# B&R Automation Studio project Agroittica (part 4)

```iecst
				intern.AsIOAccWriteValue := (51200/UINT_TO_REAL(intern.Parameters.Units_rev)) * (DINT_TO_REAL(IO_Cfg.MPGen.RefSpeed)/40.0);	(* Scale from units/s to uSteps/25ms. *)

				IF ((AsIOAccWrite_0.status = ERR_OK) AND ((intern.AsIOAccWriteValue > 65535.0) OR (intern.AsIOAccWriteValue < -65535.0) OR (* Overflow *)
	 					((IO_Cfg.MPGen.RefSpeed > 0) AND (intern.AsIOAccWriteValue < 0))) OR																					(* Positive overflow? *)
						((IO_Cfg.MPGen.RefSpeed < 0) AND (intern.AsIOAccWriteValue > 0))) THEN																				(* Negative overflow? *)

					IF ((intern.OverflowWarning > 1_00_00_00) OR (intern.OverflowWarning < 0)) THEN																	(* Already recorded 4 overflow states? *)
						intern.OverflowWarning := ((ABS(intern.OverflowWarning) + 1_00_00_00_00) * -1);																(* Make number negative and show number of overflow's occured + 4 recorded. *)
					ELSE
						intern.OverflowWarning := (intern.OverflowWarning * 100) + intern.StateMan;																		(* Recorded which step where overflow occured. *)
					END_IF

					IF (IO_Cfg.MPGen.RefSpeed > 0) THEN																																							(* Positive overflow? *)
						AsIOAccWrite_0.value := 65535;																																								(* Set to maximum. (16#FFFF = 65535) *)
					ELSIF (IO_Cfg.MPGen.RefSpeed < 0) THEN																																					(* Negitive overflow? *)
						AsIOAccWrite_0.value := -65535;																																								(* Set to maximum. (16# = -65535) *)
					END_IF

				ELSE																																																							(* Write value not overflowed. *)
					AsIOAccWrite_0.value := REAL_TO_UDINT(intern.AsIOAccWriteValue);																								(* Copy required write value. *)
				END_IF

				AsIOAccWrite_0(enable:=1, pDeviceName:=ADR(intern.IO_Mapping.DeviceName), pChannelName:=ADR(intern.ChannelName));	(* Write to register. *)

				IF (AsIOAccWrite_0.status <> ERR_FUB_BUSY) THEN																																		(* Function done? *)
					IF (AsIOAccWrite_0.status = ERR_OK) THEN																																				(* No error? *)

						IF ((Mode = 0) OR (Mode = 60) OR (intern.Cfg_State = 255)) THEN																								(* Write all configuration values to XMS module? *)
							intern.StateMan := intern.StateMan + 1;																																			(* Next XSM step. *)
						ELSE
							Done						:= 1;																																												(* Set Done flag. *)
							intern.StateMan := 0;																																												(* Wait for new command. *)
						END_IF

					ELSE																																																						(* AsIOAccRead Error? *)
						Status					:= AsIOAccWrite_0.status;																																			(* Copy AsIOAccWrite status. *)
					END_IF
				END_IF
			#endif
			#ifdef _SGC
				CASE (intern.IO_Mapping.Channel) OF
					0..1:		AsIOAccWriteReg_0.registerNr:= 68;																																			(* 1st motor channel selected. (Reg 68) *)
					2:			AsIOAccWriteReg_0.registerNr:= 132;																																			(* 2nd motor channel selected. (Reg 132) *)
					3:			AsIOAccWriteReg_0.registerNr:= 196;																																			(* 3rd motor channel selected. (Reg 196) *)
					4:			AsIOAccWriteReg_0.registerNr:= 260;																																			(* 4th motor channel selected. (Reg 260) *)
				END_CASE

				intern.AsIOAccWriteValue := (51200/UINT_TO_REAL(intern.Parameters.Units_rev)) * (DINT_TO_REAL(IO_Cfg.MPGen.RefSpeed)/40.0);	(* Scale from units/s to uSteps/25ms. *)

				IF ((AsIOAccWrite_0.status = ERR_OK) AND ((intern.AsIOAccWriteValue > 65535.0) OR (intern.AsIOAccWriteValue < -65535.0) OR (* Overflow *)
	 					((IO_Cfg.MPGen.RefSpeed > 0) AND (intern.AsIOAccWriteValue < 0))) OR																					(* Positive overflow? *)
						((IO_Cfg.MPGen.RefSpeed < 0) AND (intern.AsIOAccWriteValue > 0))) THEN																				(* Negative overflow? *)

					IF ((intern.OverflowWarning > 1_00_00_00) OR (intern.OverflowWarning < 0)) THEN																	(* Already recorded 4 overflow states? *)
						intern.OverflowWarning := ((ABS(intern.OverflowWarning) + 1_00_00_00_00) * -1);																(* Make number negative and show number of overflow's occured + 4 recorded. *)
					ELSE
						intern.OverflowWarning := (intern.OverflowWarning * 100) + intern.StateMan;																		(* Recorded which step where overflow occured. *)
					END_IF

					IF (IO_Cfg.MPGen.RefSpeed > 0) THEN																																							(* Positive overflow? *)
						AsIOAccWriteReg_0.value := 65535;																																							(* Set to maximum. (16#FFFF = 65535) *)
					ELSIF (IO_Cfg.MPGen.RefSpeed < 0) THEN																																					(* Negitive overflow? *)
						AsIOAccWriteReg_0.value := -65535;																																						(* Set to maximum. (16# = -65535) *)
					END_IF

				ELSE																																																							(* Write value not overflowed. *)
					AsIOAccWriteReg_0.value := REAL_TO_UDINT(intern.AsIOAccWriteValue);																							(* Copy required write value. *)
				END_IF

				AsIOAccWriteReg_0(enable:=1, size:=2);																																						(* Write to register. *)

				IF (AsIOAccWriteReg_0.status <> ERR_FUB_BUSY) THEN																																(* Function done? *)
					IF (AsIOAccWriteReg_0.status = ERR_OK) THEN																																			(* No error? *)

						IF ((Mode = 0) OR (Mode = 60) OR (intern.Cfg_State = 255)) THEN																								(* Write all configuration values to XMS module? *)
							intern.StateMan := intern.StateMan + 1;																																			(* Next XSM step. *)
						ELSE
							Done						:= 1;																																												(* Set Done flag. *)
							intern.StateMan := 0;																																												(* Wait for new command. *)
						END_IF

					ELSIF ((AsIOAccWriteReg_0.status = ioacERR_ACCESS) AND (intern.Retries < 2)) THEN																(* Access error? try again upto 2 times. *)
						intern.Retries:= intern.Retries + 1;																																					(* Increament retries counter. *)
					ELSE																																																						(* AsIOAccRead Error? *)
						Status					:= AsIOAccWriteReg_0.status;																																	(* Copy AsIOAccWrite status. *)
					END_IF
				END_IF
			#endif

			(* IO Configuration - Jolt time limitation. *)
			67:
				IF (IO_Cfg.MPGen.JoltTimeLimitation > 16) THEN																																		(* Jolt Time Limitation invalid? *)

					Status := 50267;																																																(* JoltTimeLimitation_Invalid *)

				ELSE

				#ifdef _SG4
					CASE (intern.IO_Mapping.Channel) OF
						0..1:		intern.ChannelName := 'JoltTime01';																																		(* 1st motor channel selected. (Reg 75) *)
						2:			intern.ChannelName := 'JoltTime02';																																		(* 2nd motor channel selected. (Reg 139) *)
						3:			intern.ChannelName := 'JoltTime03';																																		(* 3rd motor channel selected. (Reg 203) *)
						4:			intern.ChannelName := 'JoltTime04';																																		(* 4th motor channel selected. (Reg 267) *)
					END_CASE

					AsIOAccWrite_0.value := SINT_TO_UDINT(IO_Cfg.MPGen.JoltTimeLimitation);																					(* Required value. *)
					AsIOAccWrite_0(enable:=1, pDeviceName:=ADR(intern.IO_Mapping.DeviceName), pChannelName:=ADR(intern.ChannelName));	(* Write to register. *)

					IF (AsIOAccWrite_0.status <> ERR_FUB_BUSY) THEN																																	(* Function done? *)
						IF (AsIOAccWrite_0.status = ERR_OK) THEN																																			(* No error? *)
							IF ((Mode = 0) OR (Mode = 60) OR (intern.Cfg_State = 255)) THEN																							(* Module power back on? *)
								intern.Cfg_State := 1;																																										(* Reset IO Cfg Done flag. *)
							END_IF
							Done						:= 1;																																												(* Set Done flag. *)
							intern.StateMan := 0;																																												(* Wait for new command. *)
						ELSE																																																					(* AsIOAccRead Error? *)
							Status					:= AsIOAccWrite_0.status;																																		(* Copy AsIOAccWrite status. *)
						END_IF
					END_IF
				#endif
				#ifdef _SGC
					CASE (intern.IO_Mapping.Channel) OF
						0..1:		AsIOAccWriteReg_0.registerNr:= 75;																																		(* 1st motor channel selected. (Reg 75) *)
						2:			AsIOAccWriteReg_0.registerNr:= 139;																																		(* 2nd motor channel selected. (Reg 139) *)
						3:			AsIOAccWriteReg_0.registerNr:= 203;																																		(* 3rd motor channel selected. (Reg 203) *)
						4:			AsIOAccWriteReg_0.registerNr:= 267;																																		(* 4th motor channel selected. (Reg 267) *)
					END_CASE

					AsIOAccWriteReg_0.value := SINT_TO_UDINT(IO_Cfg.MPGen.JoltTimeLimitation);																			(* Required value. *)
					AsIOAccWriteReg_0(enable:=1, size:=1);																																					(* Write to register. *)

					IF (AsIOAccWriteReg_0.status <> ERR_FUB_BUSY) THEN																															(* Function done? *)
						IF (AsIOAccWriteReg_0.status = ERR_OK) THEN																																		(* No error? *)
							IF ((Mode = 0) OR (Mode = 60) OR (intern.Cfg_State = 255)) THEN																							(* Module power back on? *)
								intern.Cfg_State := 1;																																										(* Reset IO Cfg Done flag. *)
							END_IF
							Done						:= 1;																																												(* Set Done flag. *)
							intern.StateMan := 0;																																												(* Wait for new command. *)
						ELSIF ((AsIOAccWriteReg_0.status = ioacERR_ACCESS) AND (intern.Retries < 2)) THEN															(* Access error? try again upto 2 times. *)
							intern.Retries:= intern.Retries + 1;																																				(* Increament retries counter. *)
						ELSE																																																					(* AsIOAccRead Error? *)
							Status					:= AsIOAccWrite_0.status;																																		(* Copy AsIOAccWrite status. *)
						END_IF
					END_IF
				#endif

				END_IF

			(* Error handling - Check reset flag is OFF. *)
			1000:

				IF (pIO_Mapping <> 0) THEN																																												(* Address non-Zero? *)
					memcpy(ADR(intern.IO_Mapping), pIO_Mapping, SIZEOF(intern.IO_Mapping));																					(* Get update intern.IO_Mapping data. *)
				ELSE																																																							(* Error? *)
					Status := 50202;																																																(* pintern.IO_Mapping_Invalid. *)
				END_IF

				IF ((intern.Cfg_State = 255) AND (intern.IO_Mapping.ModuleOK)) THEN																								(* Module power back on? *)
					Status						:= 0;																																													(* Reset status. *)
					intern.StateMan 	:= 0;																																													(* Wait for new command. *)
				ELSIF (NOT(Reset) AND (intern.Cfg_State <> 255))THEN																															(* Reset OFF? *)
					intern.StateMan := intern.StateMan + 1;																																					(* Next XSM step. *)
				END_IF

			(* Error handling - Reset error on positve edge. *)
			1001:

				IF (Reset) THEN																																																		(* Reset / Error acknownledge? *)
					Reset							:= 0;																																													(* Reset reset. *)
					Status						:= 0;																																													(* Reset status. *)
				END_IF

				IF (NOT(Config) AND (Status = 0)) THEN																																						(* Start new configuration reset? *)
					intern.StateMan 	:= 0;																																													(* Wait for new command. *)
				END_IF

			(* Should not get here, invalid state. *)
			ELSE
				intern.StateMan := 1000;

		END_CASE

	ELSE
		intern.StateMan 	:= 0;																																																(* Wait for new command. *)
		Status := ERR_FUB_ENABLE_FALSE;																																												(* Function not enabled status. *)
	END_IF

	(********************************************************************************************************************
		!!!!!!!!!!!!!!!!!!!!!!!!!!!!!!!!!!!!!!!!! NO MORE CODE BEYOND THIS POINT !!!!!!!!!!!!!!!!!!!!!!!!!!!!!!!!!!!!!!!!!
	*********************************************************************************************************************)
END_FUNCTION_BLOCK
```

#### XSM_AcyclicRead.st - Provide alarm detail in form of BOOLEAN array for VC & User.
```iecst
FUNCTION_BLOCK XSM_AcyclicRead
	(* Implementation of XSM_AcyclicRead *)
	(********************************************************************************************************************
		Filename		: XSM_AcyclicRead.scr
		Version			: 00.01
		Date				: 14th July 2009
		Written by	: Andy Lees at B&R Industrial Automation Ltd. (UK)
		Customer		: Sheepy.
		Application : .
		Description	:	Provide alarm detail in form of BOOLEAN array for VC & User.

									Status:-

										0				ERR_OK

										50100		XSM_ModuleNotOK
										50101		XSM_ModuleID_Invalid -	X20 ->	X20SM1426 = 9857,						1x Stepper motor module 1A, 4 DI
																														X20SM1436 = 9858,						1x Stepper motor module 3A, 4 DI

																										X67 ->	X67SM2436 = 7627,						2x Stepper motor module 3A, 2x3 DI
																														X67SM4320 = 7628,						4x Stepper motor module 1A

																						ACOPOSmicro ->	80SD100XD.C0XX-01 = 42148,	2x Stepper motor 10 A, X2X, 2 Trigger Inputs.
																														80SD100XS.C0XX-01 = 42414,	1x Stepper motor 10 A, X2X, 2 DI (1 Trigger Input).
 																														80SD100XS.C04X-01 = 42880,	1x Stepper motor 10 A, X2X, 2 DI (1 Trigger Input), 1x ABR.
																														80SD100XD.C044-01 = 42881,	2x Stepper motor 10 A, X2X, 2x ABR, 2 Trigger Inputs.
																														80SD100XS.C04X-13 = 42882,	1x Stepper motor 10 A, X2X, 1x ABR, 4 DI/2 DO
																														80SD100XD.C04X-13 = 42893,	2x Stepper motor 10 A, X2X, 1x ABR, 4 DI/2 DO.
																														80SD100XD.C0XX-21 = 42894,	2x Stepper motor 10 A, X2X, 2 Inputs ±10 V.
										50109		XSM_Motor_Invalid.

										50202		pIO_Mapping_Invalid.

										50200		Read acyclic mode invalid.

										30190 - 30199 AsIOAcc

										65534		ERR_FUB_ENABLE_FALSE

									Mode:-

										1				Read DC bus voltage in V.
										2				Read Module temperature of the power output stage in °C.
										3				Read Module temperature in °C.

										4				Read Referenced zero position of the cyclic counter.
										5				Read Current position acyclic.
										6				Read Referenced zero position of the acyclic counter.

		History			: 14th July 2009		v00.01
									First release - Tested on X20CP1486 N2.95 with X20SM1426 on X2X & Ethernet Power Link.

	*********************************************************************************************************************)
	IF (Enable) THEN																																																			(* Function block enabled? *)

		(******************************************************************************************************************
			Errors force to handle errors?
		*******************************************************************************************************************)
		IF ((Status <> ERR_OK) AND (Status <> ERR_FUB_ENABLE_FALSE) AND (Status <> ERR_FUB_BUSY) AND (intern.StateMan < 1000)) THEN	(* Error and not error handling state's? *)
			intern.StateMan := 1000;																																														(* Handle errors. *)
		END_IF

		(******************************************************************************************************************
			SXM IO Configuratin state machine.
		*******************************************************************************************************************)
		CASE (intern.StateMan) OF																																															(* State machine. *)

			(* Init - Wait for command. *)
			0:
				IF ((Status = ERR_FUB_ENABLE_FALSE) OR (Status = ERR_FUB_BUSY)) THEN																							(* Clear function not enable or busy status? *)
					Status := ERR_OK;																																																(* Function OK. *)
				END_IF

				IF (pIO_Mapping <> 0) THEN																																												(* Address non-Zero? *)
					memcpy(ADR(intern.IO_Mapping), pIO_Mapping, SIZEOF(intern.IO_Mapping));																					(* Get update intern.IO_Mapping data. *)
				ELSE																																																							(* Error? *)
					Status := 50202;																																																(* pIO_Mapping_Invalid. *)
				END_IF

				IF ((intern.IO_Mapping.ModuleID <> 9857) AND (intern.IO_Mapping.ModuleID <> 9858) AND															(* Not X20SM1426, X20SM1436? *)
						(intern.IO_Mapping.ModuleID <> 7627) AND (intern.IO_Mapping.ModuleID <> 7628) AND															(* Not X67SM2436, X67SM4320? *)
						(intern.IO_Mapping.ModuleID <> 42148) AND (intern.IO_Mapping.ModuleID <> 42414) AND														(* Not 80SD100XD.C0XX-01, 80SD100XS.C0XX-01? *)
						(intern.IO_Mapping.ModuleID <> 42880) AND (intern.IO_Mapping.ModuleID <> 42881) AND														(* Not 80SD100XS.C04X-01, 80SD100XD.C044-01? *)
						(intern.IO_Mapping.ModuleID <> 42882) AND (intern.IO_Mapping.ModuleID <> 42893) AND														(* Not 80SD100XS.C04X-13, 80SD100XD.C04X-13? *)
						(intern.IO_Mapping.ModuleID <> 42894)) THEN																																		(* Not 80SD100XD.C0XX-21? *)
					Status := 50101;																																																(* Error - XSM_ModuleID_Invalid *)
				ELSIF (((intern.IO_Mapping.ModuleID = 9857) AND ((intern.IO_Mapping.Channel < 0) OR (intern.IO_Mapping.Channel > 1))) OR	(* X20SM1426 - Only 1 motor possible. *)
							 ((intern.IO_Mapping.ModuleID = 9858) AND ((intern.IO_Mapping.Channel < 0) OR (intern.IO_Mapping.Channel > 1))) OR	(* X20SM1436 - Only 1 motor possible. *)
							 ((intern.IO_Mapping.ModuleID = 7627) AND ((intern.IO_Mapping.Channel < 0) OR (intern.IO_Mapping.Channel > 2))) OR	(* X67SM2436 - Only 2 motor possible. *)
							 ((intern.IO_Mapping.ModuleID = 7628) AND ((intern.IO_Mapping.Channel < 0) OR (intern.IO_Mapping.Channel > 4)))	OR	(* X67SM4320 - Only 4 motor possible. *)
							 ((intern.IO_Mapping.ModuleID = 42148) AND ((intern.IO_Mapping.Channel < 0) OR (intern.IO_Mapping.Channel > 2))) OR	(* 80SD100XD.C0XX-01 - Only 2 motor possible. *)
							 ((intern.IO_Mapping.ModuleID = 42414) AND ((intern.IO_Mapping.Channel < 0) OR (intern.IO_Mapping.Channel > 1))) OR	(* 80SD100XS.C0XX-01 - Only 1 motor possible. *)
							 ((intern.IO_Mapping.ModuleID = 42880) AND ((intern.IO_Mapping.Channel < 0) OR (intern.IO_Mapping.Channel > 1))) OR	(* 80SD100XS.C04X-01 - Only 1 motor possible. *)
							 ((intern.IO_Mapping.ModuleID = 42881) AND ((intern.IO_Mapping.Channel < 0) OR (intern.IO_Mapping.Channel > 2))) OR	(* 80SD100XD.C044-01 - Only 2 motor possible. *)
							 ((intern.IO_Mapping.ModuleID = 42882) AND ((intern.IO_Mapping.Channel < 0) OR (intern.IO_Mapping.Channel > 1))) OR	(* 80SD100XS.C04X-13 - Only 1 motor possible. *)
							 ((intern.IO_Mapping.ModuleID = 42893) AND ((intern.IO_Mapping.Channel < 0) OR (intern.IO_Mapping.Channel > 2))) OR	(* 80SD100XD.C04X-13 - Only 2 motor possible. *)
							 ((intern.IO_Mapping.ModuleID = 42894) AND ((intern.IO_Mapping.Channel < 0) OR (intern.IO_Mapping.Channel > 2)))		(* 80SD100XD.C0XX-21 - Only 2 motor possible. *)
							) THEN																																																				(* Selected motor invalid? *)
					Status := 50109;																																																	(* XSM_Motor_Invalid? *)
				END_IF

			#ifdef _SGC
				AsIOAccReadReg_0.nodeNr:= DINT_TO_USINT(atoi(ADR(intern.IO_Mapping.DeviceName) + FIND(intern.IO_Mapping.DeviceName, 'ST') + 1));	(* Get node number on X2X. *)
			#endif

				intern.ReadOK:= (intern.ReadOK AND Read);																																				(* Detect +edge of Read. *)

				IF ((Status = ERR_OK) AND NOT(intern.ReadOK) AND (Read)) THEN																										(* Read acyclic data? *)
					intern.Retries:= 0;																																														(* Reset retries. *)
					Status := ERR_FUB_BUSY;																																												(* Function busy status. *)
					CASE (Mode) OF
						1:			intern.StateMan		:= 10;																																						(* Read DC bus voltage in V. *)
						2:			intern.StateMan 	:= 20;																																						(* Read Module temperature of the power output stage in °C. *)
						3:			intern.StateMan 	:= 30;																																						(* Read Module temperature in °C. *)
						4:			intern.StateMan 	:= 40;																																						(* Read Referenced zero position of the cyclic counter. *)
						5:			intern.StateMan 	:= 50;																																						(* Read Current position acyclic. *)
						6:			intern.StateMan 	:= 60;																																						(* Read Referenced zero position of the acyclic counter. *)
						ELSE	Status := 50400;																																											(* Read acyclic mode invalid. *)
					END_CASE
				END_IF

			(* Read DC bus voltage in V. *)
			10:
			#ifdef _SG4
				intern.ChannelName := 'UZKVoltage';																																							(* Read DC bus voltage in V. (Reg 42) *)

				AsIOAccRead_0(enable:=1, pDeviceName:=ADR(intern.IO_Mapping.DeviceName), pChannelName:=ADR(intern.ChannelName));	(* Read acyclic data. *)

				IF (AsIOAccRead_0.status <> ERR_FUB_BUSY) THEN																																	(* Function done? *)
					IF (AsIOAccRead_0.status = ERR_OK) THEN																																				(* No error? *)
						ReadData.DC_BusVoltage:= UDINT_TO_UINT(AsIOAccRead_0.value);																								(* Copy data. *)
						intern.ReadOK:= 	TRUE;																																											(* Read OK. *)
						intern.StateMan:= 0;
					ELSE																																																					(* AsIOAccRead Error? *)
						Status:= AsIOAccRead_0.status;
					END_IF
				END_IF
			#endif
			#ifdef _SGC
				AsIOAccReadReg_0.registerNr:= 42;																																								(* Read DC bus voltage in V. (Reg 42) *)

				AsIOAccReadReg_0(enable:= 1, size:= 2);																																					(* Read acyclic data. *)

				IF (AsIOAccReadReg_0.status <> ERR_FUB_BUSY) THEN																																(* Function done? *)
					IF (AsIOAccReadReg_0.status = ERR_OK) THEN																																		(* No error? *)
						ReadData.DC_BusVoltage:= UDINT_TO_UINT(AsIOAccReadReg_0.value);																							(* Update error code. *)
						intern.ReadOK:= 	TRUE;																																											(* Read OK. *)
						intern.StateMan:= 0;
					ELSIF ((AsIOAccReadReg_0.status = ioacERR_ACCESS) AND (intern.Retries < 2)) THEN															(* Access error? try again upto 2 times. *)
						intern.Retries:= intern.Retries + 1;																																				(* Increament retries counter. *)
					ELSE																																																					(* AsIOAccReadReg Error? *)
						Status:= AsIOAccReadReg_0.status;																																						(* Copy AsIOAccReadReg status. *)
					END_IF
				END_IF
			#endif

			(* Read Module temperature of the power output stage in °C. *)
			20:
			#ifdef _SG4
				intern.ChannelName := 'CoolerTemperature';																																			(* Read Module temperature of the power output stage in °C. (Reg 44) *)

				AsIOAccRead_0(enable:=1, pDeviceName:=ADR(intern.IO_Mapping.DeviceName), pChannelName:=ADR(intern.ChannelName));	(* Read acyclic data. *)

				IF (AsIOAccRead_0.status <> ERR_FUB_BUSY) THEN																																	(* Function done? *)
					IF (AsIOAccRead_0.status = ERR_OK) THEN																																				(* No error? *)
						ReadData.PowerStage_Temperature:= UDINT_TO_SINT(AsIOAccRead_0.value);																				(* Copy data. *)
						intern.ReadOK:= 	TRUE;																																											(* Read OK. *)
						intern.StateMan:= 0;
					ELSE																																																					(* AsIOAccRead Error? *)
						Status:= AsIOAccRead_0.status;
					END_IF
				END_IF
			#endif
			#ifdef _SGC
				AsIOAccReadReg_0.registerNr:= 44;																																								(* Read Module temperature of the power output stage in °C. (Reg 44). *)

				AsIOAccReadReg_0(enable:= 1, size:= 1);																																					(* Read acyclic data. *)

				IF (AsIOAccReadReg_0.status <> ERR_FUB_BUSY) THEN																																(* Function done? *)
					IF (AsIOAccReadReg_0.status = ERR_OK) THEN																																		(* No error? *)
						ReadData.PowerStage_Temperature:= UDINT_TO_SINT(AsIOAccReadReg_0.value);																		(* Update error code. *)
						intern.ReadOK:= 	TRUE;																																											(* Read OK. *)
						intern.StateMan:= 0;
					ELSIF ((AsIOAccReadReg_0.status = ioacERR_ACCESS) AND (intern.Retries < 2)) THEN															(* Access error? try again upto 2 times. *)
						intern.Retries:= intern.Retries + 1;																																				(* Increament retries counter. *)
					ELSE																																																					(* AsIOAccReadReg Error? *)
						Status:= AsIOAccReadReg_0.status;																																						(* Copy AsIOAccReadReg status. *)
					END_IF
				END_IF
			#endif

			(* Read Module temperature in °C. *)
			30:
			#ifdef _SG4
				intern.ChannelName := 'Temperature';																																						(* Read Module temperature in °C. (Reg 46) *)

				AsIOAccRead_0(enable:=1, pDeviceName:=ADR(intern.IO_Mapping.DeviceName), pChannelName:=ADR(intern.ChannelName));	(* Read acyclic data. *)

				IF (AsIOAccRead_0.status <> ERR_FUB_BUSY) THEN																																	(* Function done? *)
					IF (AsIOAccRead_0.status = ERR_OK) THEN																																				(* No error? *)
						ReadData.Module_Temperature:= UDINT_TO_SINT(AsIOAccRead_0.value);																						(* Copy data. *)
						intern.ReadOK:= 	TRUE;																																											(* Read OK. *)
						intern.StateMan:= 0;
					ELSE																																																					(* AsIOAccRead Error? *)
						Status:= AsIOAccRead_0.status;
					END_IF
				END_IF
			#endif
			#ifdef _SGC
				AsIOAccReadReg_0.registerNr:= 46;																																								(* Read Module temperature in °C. (Reg 46). *)

				AsIOAccReadReg_0(enable:= 1, size:= 1);																																					(* Read acyclic data. *)

				IF (AsIOAccReadReg_0.status <> ERR_FUB_BUSY) THEN																																(* Function done? *)
					IF (AsIOAccReadReg_0.status = ERR_OK) THEN																																		(* No error? *)
						ReadData.Module_Temperature:= UDINT_TO_SINT(AsIOAccReadReg_0.value);																				(* Update error code. *)
						intern.ReadOK:= 	TRUE;																																											(* Read OK. *)
						intern.StateMan:= 0;
					ELSIF ((AsIOAccReadReg_0.status = ioacERR_ACCESS) AND (intern.Retries < 2)) THEN															(* Access error? try again upto 2 times. *)
						intern.Retries:= intern.Retries + 1;																																				(* Increament retries counter. *)
					ELSE																																																					(* AsIOAccReadReg Error? *)
						Status:= AsIOAccReadReg_0.status;																																						(* Copy AsIOAccReadReg status. *)
					END_IF
				END_IF
			#endif

			(* Read Referenced zero position of the cyclic counter. *)
			40:
			#ifdef _SG4
				CASE (intern.IO_Mapping.Channel) OF
					0..1:		intern.ChannelName := 'RefPos01CyclicCounter';																												(* X20SM/X67SM/ACOPOSmicro 1st motor selected.(Reg 86)*)
					2:			intern.ChannelName := 'RefPos02CyclicCounter';																												(* X67SM/ACOPOSmicro 2nd motor selected. (Reg 150)*)
					3:			intern.ChannelName := 'RefPos03CyclicCounter';																												(* 3rd motor channel selected. (Reg 214) *)
					4:			intern.ChannelName := 'RefPos04CyclicCounter';																												(* 4th motor channel selected. (Reg 278) *)
				END_CASE

				AsIOAccRead_0(enable:=1, pDeviceName:=ADR(intern.IO_Mapping.DeviceName), pChannelName:=ADR(intern.ChannelName));	(* Read acyclic data. *)

				IF (AsIOAccRead_0.status <> ERR_FUB_BUSY) THEN																																	(* Function done? *)
					IF (AsIOAccRead_0.status = ERR_OK) THEN																																				(* No error? *)
						ReadData.Encoder_RefPosCyclicCounter:= UDINT_TO_DINT(AsIOAccRead_0.value);																	(* Copy data. *)
						intern.ReadOK:= 	TRUE;																																											(* Read OK. *)
						intern.StateMan:= 0;
					ELSE																																																					(* AsIOAccRead Error? *)
						Status:= AsIOAccRead_0.status;
					END_IF
				END_IF
			#endif
			#ifdef _SGC
				CASE (intern.IO_Mapping.Channel) OF
					0..1:		AsIOAccReadReg_0.registerNr:= 86;																																			(* X20SM/X67SM/ACOPOSmicro 1st motor selected.(Reg 86)*)
					2:			AsIOAccReadReg_0.registerNr:= 150;																																		(* X67SM/ACOPOSmicro 2nd motor selected. (Reg 150)*)
					3:			AsIOAccReadReg_0.registerNr:= 214;																																		(* 3rd motor channel selected. (Reg 214) *)
					4:			AsIOAccReadReg_0.registerNr:= 278;																																		(* 4th motor channel selected. (Reg 278) *)
				END_CASE

				AsIOAccReadReg_0(enable:= 1, size:= 4);																																					(* Read acyclic data. *)

				IF (AsIOAccReadReg_0.status <> ERR_FUB_BUSY) THEN																																(* Function done? *)
					IF (AsIOAccReadReg_0.status = ERR_OK) THEN																																		(* No error? *)
						ReadData.Encoder_RefPosCyclicCounter:= UDINT_TO_DINT(AsIOAccReadReg_0.value);																(* Update error code. *)
						intern.ReadOK:= 	TRUE;																																											(* Read OK. *)
						intern.StateMan:= 0;
					ELSIF ((AsIOAccReadReg_0.status = ioacERR_ACCESS) AND (intern.Retries < 2)) THEN															(* Access error? try again upto 2 times. *)
						intern.Retries:= intern.Retries + 1;																																				(* Increament retries counter. *)
					ELSE																																																					(* AsIOAccReadReg Error? *)
						Status:= AsIOAccReadReg_0.status;																																						(* Copy AsIOAccReadReg status. *)
					END_IF
				END_IF
			#endif

			(* Read Current position acyclic. *)
			50:
			#ifdef _SG4
				CASE (intern.IO_Mapping.Channel) OF
					0..1:		intern.ChannelName := 'AbsPos1ActValAcyclic';																												(* X20SM/X67SM/ACOPOSmicro 1st motor selected.(Reg 90)*)
					2:			intern.ChannelName := 'AbsPos2ActValAcyclic';																												(* X67SM/ACOPOSmicro 2nd motor selected. (Reg 154)*)
(*					3:			intern.ChannelName := 'AbsPos3ActValAcyclic';	- Not used yet *)																											(* 3rd motor channel selected. (Reg ???) *)
(*					4:			intern.ChannelName := 'AbsPos4ActValAcyclic';	- Not used yet *)																												(* 4th motor channel selected. (Reg ???) *)
				END_CASE

				AsIOAccRead_0(enable:=1, pDeviceName:=ADR(intern.IO_Mapping.DeviceName), pChannelName:=ADR(intern.ChannelName));	(* Read acyclic data. *)

				IF (AsIOAccRead_0.status <> ERR_FUB_BUSY) THEN																																	(* Function done? *)
					IF (AsIOAccRead_0.status = ERR_OK) THEN																																				(* No error? *)
						ReadData.Encoder_ActualValue:= UDINT_TO_DINT(AsIOAccRead_0.value);																					(* Copy data. *)
						intern.ReadOK:= 	TRUE;																																											(* Read OK. *)
						intern.StateMan:= 0;
					ELSE																																																					(* AsIOAccRead Error? *)
						Status:= AsIOAccRead_0.status;
					END_IF
				END_IF
			#endif
			#ifdef _SGC
				CASE (intern.IO_Mapping.Channel) OF
					0..1:		AsIOAccReadReg_0.registerNr:= 90;																																			(* X20SM/X67SM/ACOPOSmicro 1st motor selected.(Reg 90)*)
					2:			AsIOAccReadReg_0.registerNr:= 154;																																		(* X67SM/ACOPOSmicro 2nd motor selected. (Reg 150)*)
(*					3:			AsIOAccReadReg_0.registerNr:= ???;	- Not used yet *)																																		(* 3rd motor channel selected. (Reg ???) *)
(*					4:			AsIOAccReadReg_0.registerNr:= ???;	- NOT used yet *)																																		(* 4th motor channel selected. (Reg ???) *)
				END_CASE

				AsIOAccReadReg_0(enable:= 1, size:= 4);																																					(* Read acyclic data. *)

				IF (AsIOAccReadReg_0.status <> ERR_FUB_BUSY) THEN																																(* Function done? *)
					IF (AsIOAccReadReg_0.status = ERR_OK) THEN																																		(* No error? *)
						ReadData.Encoder_ActualValue:= UDINT_TO_DINT(AsIOAccReadReg_0.value);																				(* Update error code. *)
						intern.ReadOK:= 	TRUE;																																											(* Read OK. *)
						intern.StateMan:= 0;
					ELSIF ((AsIOAccReadReg_0.status = ioacERR_ACCESS) AND (intern.Retries < 2)) THEN															(* Access error? try again upto 2 times. *)
						intern.Retries:= intern.Retries + 1;																																				(* Increament retries counter. *)
					ELSE																																																					(* AsIOAccReadReg Error? *)
						Status:= AsIOAccReadReg_0.status;																																						(* Copy AsIOAccReadReg status. *)
					END_IF
				END_IF
			#endif

			(* Read Referenced zero position of the acyclic counter. *)
			60:
			#ifdef _SG4
				CASE (intern.IO_Mapping.Channel) OF
					0..1:		intern.ChannelName := 'RefPos01AcyclicCounter';																												(* X20SM/X67SM/ACOPOSmicro 1st motor selected.(Reg 94)*)
					2:			intern.ChannelName := 'RefPos02AcyclicCounter';																												(* X67SM/ACOPOSmicro 2nd motor selected. (Reg 158)*)
(*					3:			intern.ChannelName := 'RefPos03AcyclicCounter';	- Not used yet *)																											(* 3rd motor channel selected. (Reg ???) *)
(*					4:			intern.ChannelName := 'RefPos04AcyclicCounter';	- Not used yet *)																												(* 4th motor channel selected. (Reg ???) *)
				END_CASE

				AsIOAccRead_0(enable:=1, pDeviceName:=ADR(intern.IO_Mapping.DeviceName), pChannelName:=ADR(intern.ChannelName));	(* Read acyclic data. *)

				IF (AsIOAccRead_0.status <> ERR_FUB_BUSY) THEN																																	(* Function done? *)
					IF (AsIOAccRead_0.status = ERR_OK) THEN																																				(* No error? *)
						ReadData.Encoder_RefPosAcyclicCounter:= UDINT_TO_DINT(AsIOAccRead_0.value);																	(* Copy data. *)
						intern.ReadOK:= 	TRUE;																																											(* Read OK. *)
						intern.StateMan:= 0;
					ELSE																																																					(* AsIOAccRead Error? *)
						Status:= AsIOAccRead_0.status;
					END_IF
				END_IF
			#endif
			#ifdef _SGC
				CASE (intern.IO_Mapping.Channel) OF
					0..1:		AsIOAccReadReg_0.registerNr:= 94;																																			(* X20SM/X67SM/ACOPOSmicro 1st motor selected.(Reg 94)*)
					2:			AsIOAccReadReg_0.registerNr:= 158;																																		(* X67SM/ACOPOSmicro 2nd motor selected. (Reg 158)*)
(*					3:			AsIOAccReadReg_0.registerNr:= ???;	- Not used yet *)																																		(* 3rd motor channel selected. (Reg ???) *)
(*					4:			AsIOAccReadReg_0.registerNr:= ???;	- NOT used yet *)																																		(* 4th motor channel selected. (Reg ???) *)
				END_CASE

				AsIOAccReadReg_0(enable:= 1, size:= 4);																																					(* Read acyclic data. *)

				IF (AsIOAccReadReg_0.status <> ERR_FUB_BUSY) THEN																																(* Function done? *)
					IF (AsIOAccReadReg_0.status = ERR_OK) THEN																																		(* No error? *)
						ReadData.Encoder_RefPosAcyclicCounter:= UDINT_TO_DINT(AsIOAccReadReg_0.value);															(* Update error code. *)
						intern.ReadOK:= 	TRUE;																																											(* Read OK. *)
						intern.StateMan:= 0;
					ELSIF ((AsIOAccReadReg_0.status = ioacERR_ACCESS) AND (intern.Retries < 2)) THEN															(* Access error? try again upto 2 times. *)
						intern.Retries:= intern.Retries + 1;																																				(* Increament retries counter. *)
					ELSE																																																					(* AsIOAccReadReg Error? *)
						Status:= AsIOAccReadReg_0.status;																																						(* Copy AsIOAccReadReg status. *)
					END_IF
				END_IF
			#endif

			(* Check for error reset false. *)
			1000:

				IF NOT(Reset) THEN																																															(* Reset false? *)
					intern.StateMan:= 1001;																																												(* Error ack. *)
				END_IF

			(* Check for Reset & not read data request for single read only. *)
			1001:
				IF ((Status <> ERR_OK) AND (Reset)) THEN																																				(* Error? *)
					Status:= ERR_OK;																																															(* Reset set status. *)
				END_IF

				IF (NOT(Read) AND (Status = ERR_OK)) THEN																																				(* All reset? *)
					intern.StateMan:= 0;
				END_IF

		END_CASE

	ELSE
		Status := ERR_FUB_ENABLE_FALSE;																																											(* Function not enabled status. *)
	END_IF

	(********************************************************************************************************************
		!!!!!!!!!!!!!!!!!!!!!!!!!!!!!!!!!!!!!!!!! NO MORE CODE BEYOND THIS POINT !!!!!!!!!!!!!!!!!!!!!!!!!!!!!!!!!!!!!!!!!
	*********************************************************************************************************************)
END_FUNCTION_BLOCK
```

- Visualisation Logical/Hmi/Visu (not shown)

- Visualisation Logical/Hmi/Visu_T30 (not shown)

### Program Logical/Hmi/Hmi_Support

#### Variables.var
```iecst
VAR
	change_scale : BOOL := FALSE;
	Trend_max_n_disp_value : USINT := 200;
	Trend_max_value : INT := 4000;
	Trend_min_value : INT := -1100;
	Trend_reduce_n_d_value : BOOL := FALSE;
	Trend_scroll : REAL := 0.0;
	Trend_show_value : USINT := 0;
	Trend_zoom : REAL := 0.0;
END_VAR
```

#### Cyclic.st
```iecst
PROGRAM _CYCLIC
	(* Insert code here *)

	IF (change_scale) THEN
		Trend_min_value := -20;
		Trend_max_value := 150;
	ELSE
		Trend_min_value := -1100;
		Trend_max_value := 4000;
	END_IF

	CASE Trend_show_value OF

		0:
			IF (Trend_reduce_n_d_value) THEN
				Trend_show_value 		:= 10;
				Trend_reduce_n_d_value 	:= 0;
			END_IF

			Trend_max_n_disp_value := 200;
			Trend_zoom := 1;
			Trend_scroll := 1-(0.9/Trend_zoom);

		10:
			IF (Trend_reduce_n_d_value) THEN
				Trend_show_value 		:= 20;
				Trend_reduce_n_d_value 	:= 0;
			END_IF

			Trend_max_n_disp_value := 200;

			Trend_zoom := 1.5;
			Trend_scroll := 1-(0.9/Trend_zoom);

		20:
			IF (Trend_reduce_n_d_value) THEN
				Trend_show_value 		:= 30;
				Trend_reduce_n_d_value 	:= 0;
			END_IF

			Trend_max_n_disp_value := 200;

			Trend_zoom := 2;
			Trend_scroll := 1-(0.9/Trend_zoom);

		30:
			IF (Trend_reduce_n_d_value) THEN
				Trend_show_value 		:= 40;
				Trend_reduce_n_d_value 	:= 0;
			END_IF

			Trend_max_n_disp_value := 200;

			Trend_zoom := 4;
			Trend_scroll := 1-(0.9/Trend_zoom);

		40:
			IF (Trend_reduce_n_d_value) THEN
				Trend_show_value 		:= 0;
				Trend_reduce_n_d_value 	:= 0;
			END_IF

			Trend_max_n_disp_value := 200;

			Trend_zoom := 6;
			Trend_scroll := 1-(0.9/Trend_zoom);

	END_CASE;

END_PROGRAM
```

### Program Logical/IO/io_drive (IEC)

#### Cyclic.st
```iecst
PROGRAM _CYCLIC
	(* Insert code here *)

//
//	Ctr_Fasatore.inp.posizione_mst							=		glb_fas_mst.inp.PositionActualValue6064;
//	Ctr_Fasatore.inp.velocity_mst 							=  		glb_fas_mst.inp.VelocityActualValue606C;
//	Ctr_Fasatore.inp.torque_mst 							= 		glb_fas_mst.inp.TorqueActualValue_6077;
//	Ctr_Fasatore.inp.stato_mst								=  		glb_fas_mst.inp.StatusWord6041;

	glb_drv.inp.DRV_READY 								:= 		(glb_drv.inp.StatusWord6041 AND bit_0) > 0;
	glb_drv.inp.DRV_ON 									:= 		(glb_drv.inp.StatusWord6041 AND bit_1) > 0;
	glb_drv.inp.DRV_OPERATION_ENABLED 					:= 		(glb_drv.inp.StatusWord6041 AND bit_2) > 0;
	glb_drv.inp.DRV_FAULT 								:= 		(glb_drv.inp.StatusWord6041 AND bit_3) > 0;
	glb_drv.inp.DRV_VOLT_ENABLE 						:= 		(glb_drv.inp.StatusWord6041 AND bit_4) > 0;
	glb_drv.inp.DRV_QUICK_STOP 							:= 		(glb_drv.inp.StatusWord6041 AND bit_5) > 0;
	glb_drv.inp.DRV_SWITCH_ON_DISABLED 					:= 		(glb_drv.inp.StatusWord6041 AND bit_6) > 0;
	glb_drv.inp.DRV_WARNING 							:= 		(glb_drv.inp.StatusWord6041 AND bit_7) > 0;
	glb_drv.inp.DRV_REMOTE 								:= 		(glb_drv.inp.StatusWord6041 AND bit_9) > 0;
	glb_drv.inp.DRV_TARGET_REACHED 						:= 		(glb_drv.inp.StatusWord6041 AND bit_10) > 0;
	glb_drv.inp.DRV_TARGET_STATUS 						:= 		(glb_drv.inp.StatusWord6041 AND bit_11) > 0;
	glb_drv.inp.DRV_MOVE_ERROR 							:= 		(glb_drv.inp.StatusWord6041 AND bit_12) > 0;

	IF (glb_drv.out.DRV_ON_CMD) 				THEN	glb_drv.out.ContolWord6040 := glb_drv.out.ContolWord6040 OR bit_0; 		ELSE 	glb_drv.out.ContolWord6040 := glb_drv.out.ContolWord6040 AND UINT_negato_0; END_IF
	IF (glb_drv.out.DRV_ENABLE_VOLT_CMD) 		THEN	glb_drv.out.ContolWord6040 := glb_drv.out.ContolWord6040 OR bit_1; 		ELSE 	glb_drv.out.ContolWord6040 := glb_drv.out.ContolWord6040 AND UINT_negato_1; END_IF
	IF (glb_drv.out.DRV_QUICK_STOP_CMD) 		THEN	glb_drv.out.ContolWord6040 := glb_drv.out.ContolWord6040 OR bit_2; 		ELSE 	glb_drv.out.ContolWord6040 := glb_drv.out.ContolWord6040 AND UINT_negato_2; END_IF
	IF (glb_drv.out.DRV_EN_OP_CMD) 				THEN	glb_drv.out.ContolWord6040 := glb_drv.out.ContolWord6040 OR bit_3; 		ELSE 	glb_drv.out.ContolWord6040 := glb_drv.out.ContolWord6040 AND UINT_negato_3; END_IF
	IF (glb_drv.out.DRV_START_HM_NEW_PP_CMD)	THEN	glb_drv.out.ContolWord6040 := glb_drv.out.ContolWord6040 OR bit_4; 		ELSE 	glb_drv.out.ContolWord6040 := glb_drv.out.ContolWord6040 AND UINT_negato_4; END_IF
	IF (glb_drv.out.DRV_CHANGE_SET_IMM) 		THEN	glb_drv.out.ContolWord6040 := glb_drv.out.ContolWord6040 OR bit_5; 		ELSE 	glb_drv.out.ContolWord6040 := glb_drv.out.ContolWord6040 AND UINT_negato_5; END_IF
	IF (glb_drv.out.DRV_TOGGLE_ABS_REL) 		THEN	glb_drv.out.ContolWord6040 := glb_drv.out.ContolWord6040 OR bit_6; 		ELSE 	glb_drv.out.ContolWord6040 := glb_drv.out.ContolWord6040 AND UINT_negato_6; END_IF
	IF (glb_drv.out.DRV_FAULT_RESET_CMD) 		THEN	glb_drv.out.ContolWord6040 := glb_drv.out.ContolWord6040 OR bit_7; 		ELSE 	glb_drv.out.ContolWord6040 := glb_drv.out.ContolWord6040 AND UINT_negato_7; END_IF
	IF (glb_drv.out.DRV_HALT_CMD) 				THEN	glb_drv.out.ContolWord6040 := glb_drv.out.ContolWord6040 OR bit_8; 		ELSE 	glb_drv.out.ContolWord6040 := glb_drv.out.ContolWord6040 AND UINT_negato_8; END_IF

END_PROGRAM
```

### Library Logical/IO/Encoder

#### LocalFunctions.fun
```iecst
FUNCTION_BLOCK Int_to_vel
	VAR_INPUT
		Pos : DINT;
		Maxim : DINT;
	END_VAR
	VAR_OUTPUT
		Vel : REAL;
	END_VAR
	VAR
		Ton_0 : TON;
		pos_b : DINT;
		pos_a : DINT;
		Delta_pos : REAL;
	END_VAR
END_FUNCTION_BLOCK

{REDUND_ERROR} FUNCTION_BLOCK gray_to_int (*TODO: Add your comment here*) (*$GROUP=User,$CAT=User,$GROUPICON=User.png,$CATICON=User.png*)
	VAR_INPUT
		gry : {REDUND_UNREPLICABLE} ARRAY[0..11] OF BOOL;
	END_VAR
	VAR_OUTPUT
		x : {REDUND_UNREPLICABLE} DINT;
	END_VAR
	VAR
		i : SINT;
		bin : ARRAY[0..11] OF BOOL;
		New_Member : USINT;
	END_VAR
END_FUNCTION_BLOCK
```

#### Cyclic.st
```iecst
PROGRAM _CYCLIC
	(* Insert code here *)

	glb_enc_sta.b_enable     := 1;

	glb_enc_sta.bit_res := 12; 		//Risoluzione encoder
	glb_enc_sta.pinion_diam := 130; //Diametro pignone encoder
	glb_enc_sta.enc_rev := 1; 		//Rapporto riduzione tra albero ed encoder

	glb_enc_sta.words        := REAL_TO_DINT( pow(2, glb_enc_sta.bit_res));
	glb_enc_sta.enc_range    := (glb_enc_sta.pinion_diam * 3.14 * glb_enc_sta.enc_rev); (*/* 7 is the motor reduction */*)
	glb_enc_sta.res          := glb_enc_sta.enc_range / glb_enc_sta.words;    (*/* Resol. in [U] is worked out  */*)

	IF (glb_enc_sta.b_enable = 1) THEN

		(*/* Reads the data from the GRAY ABSOLUTE ENCODER */*)
		glb_enc_sta.gry[0]  := glb_io.Di.enc_sta_bit_00;
		glb_enc_sta.gry[1]  := glb_io.Di.enc_sta_bit_01;
		glb_enc_sta.gry[2]  := glb_io.Di.enc_sta_bit_02;
		glb_enc_sta.gry[3]  := glb_io.Di.enc_sta_bit_03;
		glb_enc_sta.gry[4]  := glb_io.Di.enc_sta_bit_04;
		glb_enc_sta.gry[5]  := glb_io.Di.enc_sta_bit_05;
		glb_enc_sta.gry[6]  := glb_io.Di.enc_sta_bit_06;
		glb_enc_sta.gry[7]  := glb_io.Di.enc_sta_bit_07;
		glb_enc_sta.gry[8]  := glb_io.Di.enc_sta_bit_08;
		glb_enc_sta.gry[9]  := glb_io.Di.enc_sta_bit_09;
		glb_enc_sta.gry[10] := glb_io.Di.enc_sta_bit_10;
		glb_enc_sta.gry[11] := glb_io.Di.enc_sta_bit_11;

		gray_to_int_0.gry := glb_enc_sta.gry;
		glb_enc_sta.x := gray_to_int_0.x;
		gray_to_int_0;

		IF (glb_sim = 1) THEN

			glb_enc_sta.x := glb_enc_sim.x;

		END_IF;

		Int_to_vel_0.Maxim := glb_enc_sta.words;
		Int_to_vel_0.Pos := glb_enc_sta.x;
		Int_to_vel_0;

		IF ((glb_enc_sta.x < 0) OR (glb_enc_sta.x >= glb_enc_sta.words)) THEN
			glb_enc_sta.error := 1;
		ELSE
			glb_enc_sta.error := 0;
		END_IF
	END_IF

	//	STP_01_Vel := Int_to_vel_0.Vel;
	STP_01_Vel := 7000;
	STP_01_Pos := Int_to_vel_0.Pos;

END_PROGRAM
```

#### gray_to_int.st
```iecst
(* TODO: Add your comment here *)
FUNCTION_BLOCK gray_to_int

	bin[11] := gry[11];
	i := 0;
	x := 0;

	FOR i := 10 TO 0 BY -1 DO

		bin[i] := ((bin[i+1]) XOR (gry[i]));

	END_FOR;

	FOR i := 11 TO 0 BY -1 DO

		x := x + (bin[i] * REAL_TO_DINT( pow(2, i)));

	END_FOR;

END_FUNCTION_BLOCK

FUNCTION_BLOCK Int_to_vel

	pos_b := Pos;
	Ton_0.IN := 1;

	IF (Ton_0.Q) THEN
		Ton_0.IN := 0;

		Delta_pos := pos_b - pos_a;

		Delta_pos := SQRT(pow(Delta_pos, 2));

		IF (pos_a > pos_b) THEN

			Delta_pos := pos_b + (Maxim - pos_a);

			Delta_pos := SQRT(pow(Delta_pos, 2));

			Vel := (Delta_pos)/0.408;
		ELSE
			Vel := Delta_pos / 0.408;
		END_IF

		pos_a := pos_b;

	END_IF

	Ton_0;
	Ton_0.PT := T#400ms;

END_FUNCTION_BLOCK
```

### Program Logical/IO/Laser_Enc

#### Variables.var
```iecst
VAR
	old : REAL := 0.0;
END_VAR
```

#### Cyclic.st
```iecst
PROGRAM _CYCLIC
	(* Insert code here *)

//	Enc_laser_dist_raw;

	m_laser_enc := (2150);
	m_laser_enc := m_laser_enc / (32767-3277);

	glb_io.Ai.Enc_laser_dist_conv := ((m_laser_enc*(INT_TO_REAL (glb_io.Ai.Enc_laser_dist_raw-3277))) + Enc_laser_offset);

	glb_io.Ai.Enc_laser_dist_conv1 := ((m_laser_enc*(INT_TO_REAL (glb_io.Ai.Enc_laser_dist_raw-3277))) + Enc_laser_offset);

//	Enc_laser_dist_conv := ((2300-150)/(32767 - 3277))*((INT_TO_REAL (Enc_laser_dist_raw)) - 3277);

	IF (((glb_io.Ai.Enc_laser_dist_conv - 2) < Ricette.Laser_trigger) AND (NOT(glb_fish_shot_ons)))  THEN
		glb_io.Di.Finecorsa  := 1;
		glb_fish_shot_ons    := 1;
	END_IF;

	IF ((glb_io.Ai.Enc_laser_dist_conv > 390) AND (glb_fish_shot_ons)) THEN
		glb_fish_shot_ons := 0;
		glb_io.Di.Finecorsa  := 0;
	END_IF;
	IF (glb_io.Ai.Enc_laser_dist_conv < old) THEN
		old := glb_io.Ai.Enc_laser_dist_conv;
		END_IF;

END_PROGRAM
```

#### Init.st
```iecst
PROGRAM _INIT
	(* Insert code here *)
	glb_fish_shot_ons    := 0;

END_PROGRAM
```

### Program Logical/Axis/Program (IEC)

#### Cyclic.ld - Cyclic code
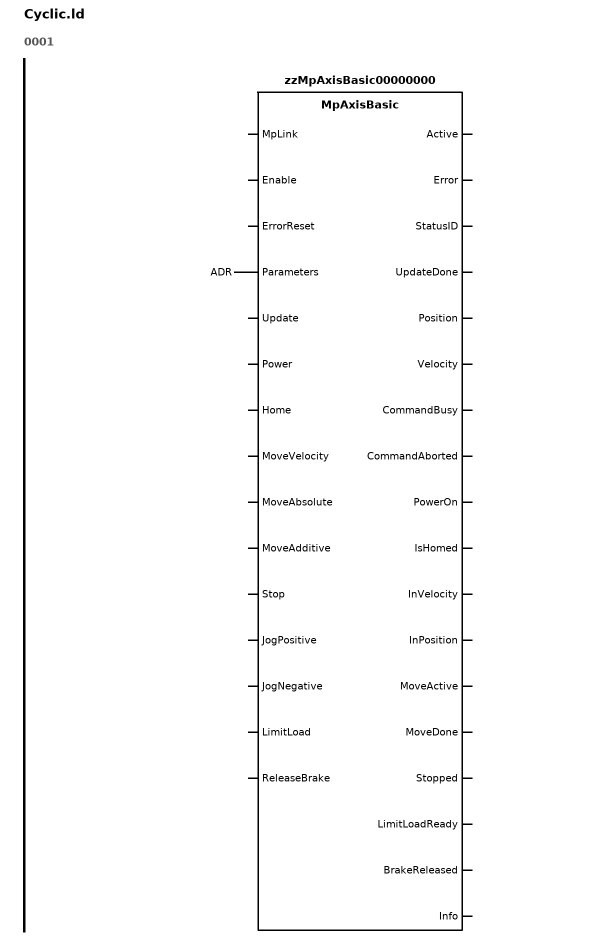
Ladder, written as Structured Text:
```iecst
PROGRAM _CYCLIC
(* Network 1 *)
zzMpAxisBasic00000000(Parameters := ADR());
END_PROGRAM
```

### Program Logical/Tcp_ip/TCP_IP (IEC)

#### Types.typ
```iecst
TYPE
	History_Buffer_typ : 	STRUCT
		state_not_changed : BOOL;
		state_name_19 : STRING[31];
		state_name_18 : STRING[31];
		state_name_17 : STRING[31];
		state_name_16 : STRING[31];
		state_name_15 : STRING[31];
		state_name_14 : STRING[31];
		state_name_13 : STRING[31];
		state_name_12 : STRING[31];
		state_name_11 : STRING[31];
		state_name_10 : STRING[31];
		state_name_9 : STRING[31];
		state_name_8 : STRING[31];
		state_name_7 : STRING[31];
		state_name_6 : STRING[31];
		state_name_5 : STRING[31];
		state_name_4 : STRING[31];
		state_name_3 : STRING[31];
		state_name_2 : STRING[31];
		state_name_1 : STRING[31];
		state_name_0 : STRING[31];
	END_STRUCT;
	Client_typ : 	STRUCT  (*TCP Client Variables*)
		sStep : UINT; (*TCP Client Step Variable*)
		TcpOpen_0 : TcpOpen; (*AsTCP.TcpOpen FUB*)
		TcpClient_0 : TcpClient; (*AsTCP.TcpClient FUB*)
		TcpRecv_0 : TcpRecv; (*AsTCP.TcpRecv FUB*)
		TcpSend_0 : TcpSend; (*AsTCP.TcpSend FUB*)
		TcpIoctl_0 : TcpIoctl; (*AsTCP.TcpIoctl FUB*)
		TcpClose_0 : TcpClose; (*AsTCP.TcpClose FUB*)
		linger_opt : tcpLINGER_typ; (*AsTCP.tcpLINGER_typ*)
		recv_timeout : UDINT; (*receive timeout*)
		connected : BOOL; (*a 1 se connesso*)
	END_STRUCT;
	Buffer_typ : 	STRUCT
		machine_in_auto : BOOL;
		machine_in_man : BOOL;
		machine_stopped : BOOL;
		machine_in_error : BOOL;
		last_cycle_request : BOOL;
		stop_request : BOOL;
		reserve1 : BOOL;
		reserve2 : BOOL;
		reserve3 : BOOL;
		client_id : USINT;
		stacksize : USINT;
		reserve6 : USINT;
		reserve4 : USINT;
		keep_alive : UDINT;
	END_STRUCT;
	TCP_typ : 	STRUCT  (*Datatyp for global Variables*)
		receive_data : Buffer_typ; (*Data which has been received*)
		send_data : Buffer_typ; (*Data which should be sent*)
		bisAlive : BOOL;
	END_STRUCT;
END_TYPE
```

#### Variables.var
```iecst
VAR
	HMI : USINT := 0;
	History_Buffer : History_Buffer_typ := (0);
	Client : Client_typ := (0); (*Data for Client Task*)
	buffer : TCP_typ;
END_VAR
```

#### Cyclic.st
```iecst
PROGRAM _CYCLIC
	HMI := 1;

	IF (Eth_connect.disable = 1) THEN Client.sStep := 40; RETURN;
	END_IF

	(* DATA TO SEND*)
	buffer.send_data.keep_alive 		:= buffer.send_data.keep_alive + 1; 								(* Generate a "running" variable for Data transfer *)
	buffer.send_data.machine_in_auto 	:= Eth_connect.machine_in_auto;
	buffer.send_data.machine_in_man  	:= Eth_connect.machine_in_man;
	buffer.send_data.machine_stopped 	:= Eth_connect.machine_stopped;
	buffer.send_data.machine_in_error	:= Eth_connect.machine_in_error;

//	IF 	  strcmp(ADR(glb_nome_macchina), ADR("P01056")) = 0 THEN
//		buffer.send_data.client_id := 1;
//	ELSIF strcmp(ADR(glb_nome_macchina), ADR("P01057")) = 0 THEN
//		buffer.send_data.client_id := 2;
//	ELSIF strcmp(ADR(glb_nome_macchina), ADR("P01058")) = 0 THEN
//		buffer.send_data.client_id := 3;
//	ELSIF strcmp(ADR(glb_nome_macchina), ADR("P01059")) = 0 THEN
//		buffer.send_data.client_id := 4;
//	ELSIF strcmp(ADR(glb_nome_macchina), ADR("P01183")) = 0 THEN
//		buffer.send_data.client_id := 5;
//	END_IF

	(* DATA RECEIVED *)
	Eth_connect.stop_request 			:= buffer.receive_data.stop_request;
	Eth_connect.last_cycle_request 		:= buffer.receive_data.last_cycle_request;

	(* AZZERO GLI STATI DEL PROTOCOLLO DI COMUNICAZIONE E DELLA LIBRERIA TCP *)
	Eth_connect.protocol_state.place_older      := 1;

	Eth_connect.tcp_state.tcpclient 			:= 1;
	Eth_connect.tcp_state.tcpclose  			:= 1;
	Eth_connect.tcp_state.tcperror 				:= 1;
	Eth_connect.tcp_state.tcpioctl  			:= 1;
	Eth_connect.tcp_state.tcpopen   			:= 1;
	Eth_connect.tcp_state.tcprecv   			:= 1;
	Eth_connect.tcp_state.tcpsend   			:= 1;

	(* TCP COMUNICATION PROGRAM *)
	CASE Client.sStep OF

		0: (* Open Ethernet Interface *)
			Eth_connect.tcp_state.tcpopen := 0;
			Client.TcpOpen_0.enable := 1;
			Client.TcpOpen_0.pIfAddr := 0;  (* Which Interface to open *)
			Client.TcpOpen_0.port := 12001;  (* Port on client side to use *)
			Client.TcpOpen_0.options := 0;
			Client.TcpOpen_0;  (* Call the Function *)
			Eth_connect.no_comunication := 1;

			IF Client.TcpOpen_0.status = 0 THEN  (* TcpOpen successfull *)
				Client.sStep := 5;
			ELSIF Client.TcpOpen_0.status = ERR_FUB_BUSY THEN  (* TcpOpen not finished -> redo *)
				(* Busy *)
			ELSE  (* Goto Error Step *)
				Client.sStep := 100;
				buffer.send_data.keep_alive := 0; (* Reset the counter *)
			END_IF

		5:
			Eth_connect.tcp_state.tcpioctl := 0;
			Client.linger_opt.lLinger := 0; (* linger Time = 0 *)
			Client.linger_opt.lOnOff := 1; (* linger Option ON *)

			Client.TcpIoctl_0.enable := 1;
			Client.TcpIoctl_0.ident := Client.TcpOpen_0.ident; (* Connection Ident from AsTP.TCP_Open *)
			Client.TcpIoctl_0.ioctl := tcpSO_LINGER_SET; (* Set Linger Options *)
			Client.TcpIoctl_0.pData := ADR(Client.linger_opt);
			Client.TcpIoctl_0.datalen := SIZEOF(Client.linger_opt);
			Client.TcpIoctl_0;

			IF Client.TcpIoctl_0.status = 0 THEN  (* TcpIoctl successfull *)
				Client.sStep := 10;
			ELSIF Client.TcpIoctl_0.status = ERR_FUB_BUSY THEN  (* TcpIoctl not finished -> redo *)
				(* Busy *)
			ELSE  (* Goto Error Step *)
				Client.sStep := 100;
				buffer.send_data.keep_alive := 0; (* Reset the counter *)
			END_IF

		10: (* Connect to the other Station *)
			Eth_connect.tcp_state.tcpclient := 0;
			Client.TcpClient_0.enable := 1;
			Client.TcpClient_0.ident := Client.TcpOpen_0.ident;  (* Connection Ident from AsTCP.TCP_Open *)
			Client.TcpClient_0.portserv := 12000;  (* Port on server side to use *)
			Client.TcpClient_0.pServer := (*ADR('192.168.250.15');*) ADR(Eth_connect.Server_Ip_Add);  (* Server Address *)
			Client.TcpClient_0;  (* Call the Function*)

			IF Client.TcpClient_0.status = 0 THEN  (* Open ok -> Send Data *)
				Client.sStep := 20;
			ELSIF Client.TcpClient_0.status = ERR_FUB_BUSY THEN  (* TcpClient not finished -> redo *)
				(* Busy *)
			ELSIF Client.TcpClient_0.status = tcpERR_INVALID THEN  (* Port error -> Close actual connection, and reopen a new one *)
				Client.sStep := 40;
			ELSE  (* Goto Error Step *)
				Client.sStep := 100;
				buffer.send_data.keep_alive := 0; (* Reset the counter *)
			END_IF

		20: (* Send Data to the Server *)
			Eth_connect.tcp_state.tcpsend := 0;
			Client.TcpSend_0.enable := 1;
			Client.TcpSend_0.ident := Client.TcpOpen_0.ident;  (* Connection Ident from AsTCP.TCP_Open *)
			Client.TcpSend_0.pData := ADR(buffer.send_data);  (* Which data to send *)
			Client.TcpSend_0.datalen := SIZEOF(buffer.send_data);  (* Lenght of data to send *)
			Client.TcpSend_0.flags := 0;
			Client.TcpSend_0;  (* Call the Function*)
			Eth_connect.no_comunication := 0;

			IF Client.TcpSend_0.status = 0 THEN  (* Data was sent sucessfully -> receive data *)
				Client.sStep := 30;
			ELSIF Client.TcpSend_0.status = ERR_FUB_BUSY THEN  (* TcpSend not finished -> redo *)
				(* Busy *)
			ELSIF (Client.TcpSend_0.status = tcpERR_SENTLEN) OR (Client.TcpSend_0.status = tcpERR_NOT_CONNECTED) THEN (* Connection Lost *)
				Client.sStep := 40;
			ELSE  (* Goto Error Step *)
				Client.sStep := 100;
				buffer.send_data.keep_alive := 0; (* Reset the counter *)
			END_IF

		30: (* Receive Data from the Server *)
			Eth_connect.tcp_state.tcprecv := 0;
			Client.TcpRecv_0.enable := 1;
			Client.TcpRecv_0.ident := Client.TcpOpen_0.ident;  (* Connection Ident from AsTCP.TCP_Open *)
			Client.TcpRecv_0.pData	:= ADR(buffer.receive_data);  (* Where to store the incoming data *)
			Client.TcpRecv_0.datamax := SIZEOF(buffer.receive_data);  (* Lenght of data buffer *)
			Client.TcpRecv_0.flags := 0;
			Client.TcpRecv_0;  (* Call the Function*)
			Eth_connect.no_comunication := 0;

			IF Client.TcpRecv_0.status = 0 THEN  (* Data was received sucessfully -> Send next packet *)
				Client.sStep := 20;
				Client.recv_timeout := 0;
			ELSIF Client.TcpRecv_0.status = tcpERR_NO_DATA THEN  (* No data received - wait *)
				Client.recv_timeout := Client.recv_timeout + 1;
				IF Client.recv_timeout > 50 THEN
					Client.sStep := 40;
					Client.recv_timeout := 0;
				END_IF
				(* No Data received *)
			ELSIF Client.TcpRecv_0.status = ERR_FUB_BUSY THEN  (* TcpRecv not finished -> redo *)
				(* Busy *)
			ELSIF Client.TcpSend_0.status = tcpERR_NOT_CONNECTED THEN (* Connection Lost *)
				Client.sStep := 40;
			ELSE  (* Goto Error Step *)
				Client.sStep := 100;
				buffer.send_data.keep_alive := 0; (* Reset the counter *)
			END_IF

		40: (* Close connection *)
			Eth_connect.tcp_state.tcpclose := 0;
			Client.TcpClose_0.enable := 1;
			Client.TcpClose_0.ident := Client.TcpOpen_0.ident;  (* Connection Ident from AsTCP.TCP_Open *)
			Client.TcpClose_0.how := 0;
			Client.TcpClose_0;  (* Call the Function*)

			IF Client.TcpClose_0.status = 0 THEN  (* Close sucessfull -> Reopen the interface *)
				Client.sStep := 0;
			ELSIF Client.TcpClose_0.status = ERR_FUB_BUSY THEN  (* TcpClose not finished -> redo *)
				(* Busy *)
			ELSE  (* Goto Error Step *)
				Client.sStep := 0; // era 100
				buffer.send_data.keep_alive := 0; (* Reset the counter *)
			END_IF

		100: (* Here some error Handling has to be implemented *)
			Eth_connect.tcp_state.tcperror := 0;
			Eth_connect.no_comunication := 1;
			IF buffer.send_data.keep_alive >  1250 THEN 	(* 1250 * 4ms = 5 seconds *)
				IF (Client.TcpOpen_0.status = 32602)  THEN
					Client.sStep := 40;
				ELSE
					Client.sStep := 40; // was 0
				END_IF
			END_IF

	END_CASE

END_PROGRAM
```

#### Init.st
```iecst
PROGRAM _INIT
	(* Insert code here *)
END_PROGRAM
```

### Program Logical/main/Main (IEC)

- Visualisation Logical/main/Main/Hmi/Visu_t30 (not shown)

#### Cyclic.st - Cyclic code
```iecst
PROGRAM _CYCLIC
	(* Insert code here *)

	CASE Status OF

		STOP:
			IF glb_io.Di.Automatic AND glb_io.Di.Start THEN
				Status := AUTO;

			ELSIF NOT glb_io.Di.Automatic AND glb_io.Di.Start THEN
				Status := MANUAL;

			END_IF

		AUTO:
			IF glb_io.Di.Stop THEN
				Status := STOP;
				last_cycle := 1;
			END_IF

		MANUAL:
			IF glb_io.Di.Stop THEN
				Status := STOP;
			END_IF
		ERR:

	END_CASE;

	IF St_Gun = 0 THEN last_cycle := 0;	END_IF

	IF ((Status <> AUTO) AND (NOT last_cycle)) THEN St_Gun := 0; END_IF

	CASE St_Gun OF

		0:	// idle
			TON_01.IN 		:= 0;
			TON_02.IN 		:= 0;

			IF glb_io.Di.Si_01 THEN St_Gun := 10; END_IF

		10:	//

			TON_01.IN := 1;

			IF TON_01.Q THEN St_Gun := 20; END_IF

		20:
			glb_io.Do.Piston_up := 1;
			IF glb_io.Di.Finecorsa THEN St_Gun := 30; END_IF

		30: //shoot
			glb_io.Do.Piston_gun_1 := 1;
			TON_02.IN := 1;

			IF TON_02.Q THEN St_Gun := 40; END_IF

		40:
			IF NOT glb_io.Di.Si_01 THEN St_Gun := 50; END_IF

		50: // end & reset
			TON_01.IN 				:= 0;
			TON_02.IN 				:= 0;
			glb_io.Do.Piston_gun_1 	:= 0;
			glb_io.Do.Piston_up		:= 0;
			St_Gun 					:= 0;

	END_CASE;

	TON_01;
	TON_02;
	TON_03;

	TON_01.PT := T#1s;
	TON_02.PT := T#1s;
	TON_03.PT := T#1s;

END_PROGRAM
```

#### Variables.var - Local variables
```iecst
VAR
	last_cycle : BOOL;
	TON_03 : TON;
	TON_02 : TON;
	TON_01 : TON;
	St_Gun : USINT;
END_VAR
```

#### LocalFunctions.fun - not listed in the package file held
```iecst
{REDUND_ERROR} FUNCTION_BLOCK gun (*TODO: Add your comment here*) (*$GROUP=User,$CAT=User,$GROUPICON=User.png,$CATICON=User.png*)
	VAR_INPUT
		Peso_ok : BOOL;
		trigger_sensor : BOOL;
		finecorsa : BOOL;
		PT_pist_Delay : TIME;
		PT_end_stop : TIME;
		PT_piston_up : TIME;
		PT_trigger_gun : TIME;
	END_VAR
	VAR_OUTPUT
		end : BOOL;
		gun_out : BOOL;
		Ready : BOOL;
		Piston_down : BOOL;
		Piston_up : BOOL;
		Piston_out : BOOL;
		Clear_weight : BOOL;
	END_VAR
	VAR
		TON_08 : TON;
		TON_04 : TON;
		TON_03 : TON;
		TON_02 : TON;
		TON_01 : TON;
		St_Gun : USINT;
	END_VAR
END_FUNCTION_BLOCK
```

#### gun.st - not listed in the package file held
```iecst
FUNCTION_BLOCK gun

	CASE St_Gun OF

		0:	// idle/start
			TON_01.IN 		:= 0;
			TON_02.IN 		:= 0;

			Ready 			:= 1;

			IF (trigger_sensor) THEN St_Gun := 10;	END_IF;

		10:	// start of TON_01 timer(timer that commands the main piston)
			Ready 		:= 0;
			TON_01.IN 	:= 1;

			IF TON_01.Q THEN St_Gun := 20; END_IF;

		20: // Main Piston up
			Ready 		:= 0;
			Piston_up 	:= 1;
			//start timer delays shot
			TON_08.IN 	:= 1;

			IF (finecorsa AND (PT_piston_up = 0)) OR (TON_08.Q AND (PT_piston_up > 0)) THEN
				TON_08.IN 	:= 0;
				St_Gun 		:= 30;
			END_IF;

		30: //shoot
			Ready := 0;
			IF Peso_ok THEN gun_out := 1; END_IF;

			TON_02.IN := 1;

			IF TON_02.Q THEN
				Piston_up 		:= 0;
				Piston_down		:= 1;
				finecorsa		:= 0;
				St_Gun 			:= 40;
			END_IF;

		40:
			Ready 			:= 0;
			TON_03.IN 		:= 1;
			end 			:= 1;

			IF((NOT trigger_sensor) AND TON_03.Q) THEN
				Clear_weight	:= 1;
				St_Gun 	:= 50;
				end 	:= 0;
			END_IF;

		50: // end & reset
			Ready := 0;
			TON_01.IN 				:= 0;
			TON_02.IN 				:= 0;
			TON_03.IN 				:= 0;
			TON_04.IN				:= 0;
			TON_08.IN				:= 0;
			gun_out 				:= 0;
			Piston_out				:= 0;
			Piston_down				:= 0;
			Clear_weight			:= 0;
			St_Gun 					:= 0;
			end 					:= 0;

	END_CASE;

	TON_01;
	TON_02;
	TON_03;
	TON_04;
	TON_08;

	TON_01.PT := PT_pist_Delay;			//tempo delay pistone sollevamento pesce
	//PT_pist_Delay := T#1000ms;		//MOD FOR TEST 06/05/2025
	//TON_01.PT 		:= T#10000ms;	//MOD FOR TEST 10/12/2024
	IF (PT_trigger_gun > 0) THEN
		TON_02.PT 	:= PT_trigger_gun;
	ELSE
		TON_02.PT 	:= T#50ms; 			// tempo discesa pist soll
	END_IF
	TON_03.PT 		:= PT_end_stop;		// tempo di attesa alla fine del ciclo
	TON_04.PT 		:= T#1000ms;		// Sicurezza pistone soll
	TON_08.PT 		:= PT_piston_up;	// Se imposto questo tempo il ritorno del pistone è comandato da questo timer + il tempo della pistola (ton_2)
//	TON_08.PT 		:= T#10000ms;		//MOD FOR TEST 09/12/2024

END_FUNCTION_BLOCK
```

### Program Logical/main/Buffer_RPT (IEC)

#### Cyclic.st - Cyclic code
```iecst
PROGRAM _CYCLIC
	(* Insert code here *)
	Str_Length 	:= LEN(Eth_connect.Marel_Weight);
	Str_weight 	:= MID(Eth_connect.Marel_Weight, (Str_Length-2), 2);

	// .......................... sensore pistola ..........................
	IF(glb_io.Di.Si_01 AND (NOT s01_b))THEN
		//rpt
		RPT_Buffer.sensore_pistola[indice] := glb_io.Di.Si_01;
		RPT_Buffer.time_stamp[indice] := glb_time;
		// hmi
		sensore_pistola := 80;

		indice := indice + 1;
		updt_hmi_trend := 1;

		s01_b := TRUE;
	ELSIF((NOT glb_io.Di.Si_01) AND s01_b) THEN
		//rpt
		RPT_Buffer.sensore_pistola[indice] := glb_io.Di.Si_01;
		RPT_Buffer.time_stamp[indice] := glb_time;
		//hmi
		sensore_pistola := 0;

		indice := indice + 1;
		updt_hmi_trend := 1;

		s01_b := FALSE;
	END_IF

	// .......................... pistone sollevamento principale ..........................
	IF(glb_io.Do.Main_Piston_Up AND (NOT Piston_Up_b))THEN
		//rpt
		RPT_Buffer.pistone_soll_su[indice] := glb_io.Do.Main_Piston_Up;
		RPT_Buffer.pistone_soll_giu[indice] := glb_io.Do.Main_Piston_Down;
		RPT_Buffer.time_stamp[indice] := glb_time;
		//hmi
		pistone_soll_su := 110;
		pistone_soll_giu := 0;

		indice := indice + 1;
		updt_hmi_trend := 1;

		Piston_Up_b := TRUE;
	ELSIF((NOT glb_io.Do.Main_Piston_Up) AND Piston_Up_b) THEN
		//rpt
		RPT_Buffer.pistone_soll_su[indice] := glb_io.Do.Main_Piston_Up;
		RPT_Buffer.pistone_soll_giu[indice] := glb_io.Do.Main_Piston_Down;
		RPT_Buffer.time_stamp[indice] := glb_time;
		//hmi
		pistone_soll_su := 0;
		pistone_soll_giu := 110;

		indice := indice + 1;
		updt_hmi_trend := 1;

		Piston_Up_b := FALSE;
	END_IF

	// .......................... pistone pistola 1 ..........................
	IF(glb_io.Do.Piston_gun_1 AND (NOT gun_1_b))THEN
		//rpt
		RPT_Buffer.pistone_pistola_1[indice] := glb_io.Do.Piston_gun_1;
		RPT_Buffer.time_stamp[indice] := glb_time;
		//hmi
		pistone_pistola_1 := 140;

		indice := indice + 1;
		updt_hmi_trend := 1;

		gun_1_b := TRUE;
	ELSIF((NOT glb_io.Do.Piston_gun_1) AND gun_1_b) THEN
		//rpt
		RPT_Buffer.pistone_pistola_1[indice] := glb_io.Do.Piston_gun_1;
		RPT_Buffer.time_stamp[indice] := glb_time;
		//hmi
		pistone_pistola_1 := 0;

		indice := indice + 1;
		updt_hmi_trend := 1;
		gun_1_b := FALSE;
	END_IF

	// .......................... pistone pistola 2 ..........................
	IF(glb_io.Do.Piston_gun_2 AND (NOT gun_2_b))THEN
		//rpt
		RPT_Buffer.pistone_pistola_2[indice] := glb_io.Do.Piston_gun_2;
		RPT_Buffer.time_stamp[indice] := glb_time;
		//hmi
		pistone_pistola_2 := 140;

		indice := indice + 1;
		updt_hmi_trend := 1;
		gun_2_b := TRUE;
	ELSIF((NOT glb_io.Do.Piston_gun_2) AND gun_2_b) THEN
		//rpt
		RPT_Buffer.pistone_pistola_2[indice] := glb_io.Do.Piston_gun_2;
		RPT_Buffer.time_stamp[indice] := glb_time;
		//hmi
		pistone_pistola_2 := 0;

		indice := indice + 1;
		updt_hmi_trend := 1;
		gun_2_b := FALSE;
	END_IF

	// .......................... bilancia ..........................
	IF(glb_rpt) OR Test THEN
		//rpt
		RPT_Buffer.bilancia[indice] := Eth_connect.Marel_Weight;
		RPT_Buffer.time_stamp[indice] := glb_time;
		//hmi
		Bilancia := (STRING_TO_REAL(Str_weight));
		Bilancia := (Bilancia * INT_TO_REAL(1000));

		indice := indice + 1;
		updt_hmi_trend := 1;
		glb_rpt := FALSE;
		Test:= 0;
	END_IF

	// .......................... passo i dati al RPT_CSV ..........................
	IF (indice >= 200) THEN
		FOR i := 0 TO 199 DO
			glb_data.bilancia[i]			:= RPT_Buffer.bilancia[i];
			glb_data.pistone_pistola_1[i]	:= RPT_Buffer.pistone_pistola_1[i];
			glb_data.pistone_pistola_2[i]	:= RPT_Buffer.pistone_pistola_2[i];
			glb_data.pistone_soll_giu[i]	:= RPT_Buffer.pistone_soll_giu[i];
			glb_data.pistone_soll_su[i]		:= RPT_Buffer.pistone_soll_su[i];
			glb_data.sensore_pistola[i]		:= RPT_Buffer.sensore_pistola[i];
			glb_data.time_stamp[i]			:= RPT_Buffer.time_stamp[i];

			RPT_Buffer.bilancia[i] 			:= '0';
			RPT_Buffer.pistone_pistola_1[i]	:= 255;
			RPT_Buffer.pistone_pistola_2[i]	:= 255;
			RPT_Buffer.pistone_soll_giu[i]	:= 255;
			RPT_Buffer.pistone_soll_su[i]	:= 255;
			RPT_Buffer.sensore_pistola[i]	:= 255;
			RPT_Buffer.time_stamp[i]		:= DT#1970-01-01-00:00:00;
		END_FOR;

		FOR i := 200 TO 249 DO
			IF (RPT_Buffer.time_stamp[i] <> DT#1970-01-01-00:00:00) THEN
				RPT_Buffer.bilancia[i-200] 			:= RPT_Buffer.bilancia[i];
				RPT_Buffer.pistone_pistola_1[i-200]	:= RPT_Buffer.pistone_pistola_1[i];
				RPT_Buffer.pistone_pistola_2[i-200]	:= RPT_Buffer.pistone_pistola_2[i];
				RPT_Buffer.pistone_soll_giu[i-200]	:= RPT_Buffer.pistone_soll_giu[i];
				RPT_Buffer.pistone_soll_su[i-200]	:= RPT_Buffer.pistone_soll_su[i];
				RPT_Buffer.sensore_pistola[i-200]	:= RPT_Buffer.sensore_pistola[i];
				RPT_Buffer.time_stamp[i-200]		:= RPT_Buffer.time_stamp[i];

				RPT_Buffer.bilancia[i] 			:= '0';
				RPT_Buffer.pistone_pistola_1[i]	:= 255;
				RPT_Buffer.pistone_pistola_2[i]	:= 255;
				RPT_Buffer.pistone_soll_giu[i]	:= 255;
				RPT_Buffer.pistone_soll_su[i]	:= 255;
				RPT_Buffer.sensore_pistola[i]	:= 255;
				RPT_Buffer.time_stamp[i]		:= DT#1970-01-01-00:00:00;
			END_IF
		END_FOR

		glb_data.Trigger := 1;
		indice := 0;
	END_IF

	IF (updt_hmi_trend AND trend_enable) THEN
		Hmi_trend_01.INWrite := 1;
		Hmi_trend_02.INWrite := 1;
		Hmi_trend_03.INWrite := 1;
		Hmi_trend_04.INWrite := 1;
		Hmi_trend_05.INWrite := 1;
		Hmi_trend_06.INWrite := 1;
	ELSE
		Hmi_trend_01.INWrite := 0;
		Hmi_trend_02.INWrite := 0;
		Hmi_trend_03.INWrite := 0;
		Hmi_trend_04.INWrite := 0;
		Hmi_trend_05.INWrite := 0;
		Hmi_trend_06.INWrite := 0;
	END_IF

	updt_hmi_trend := 0;

	Hmi_trend_01.DataIn := Bilancia;
	Hmi_trend_02.DataIn := pistone_pistola_1;
	Hmi_trend_03.DataIn := pistone_pistola_2;
	Hmi_trend_04.DataIn := pistone_soll_su;
	Hmi_trend_05.DataIn := pistone_soll_giu;
	Hmi_trend_06.DataIn := sensore_pistola;

	Hmi_trend_01;
	Hmi_trend_02;
	Hmi_trend_03;
	Hmi_trend_04;
	Hmi_trend_05;
	Hmi_trend_06;

	RPT_Buffer_hmi.bilancia 			:= Hmi_trend_01.Buffer;
	RPT_Buffer_hmi.pistone_pistola_1 	:= Hmi_trend_02.Buffer;
	RPT_Buffer_hmi.pistone_pistola_2 	:= Hmi_trend_03.Buffer;
	RPT_Buffer_hmi.pistone_soll_su 		:= Hmi_trend_04.Buffer;
	RPT_Buffer_hmi.pistone_soll_giu 	:= Hmi_trend_05.Buffer;
	RPT_Buffer_hmi.sensore_pistola 		:= Hmi_trend_06.Buffer;

	RPT_Buffer_hmi.bilancia[200] 			:= RPT_Buffer_hmi.bilancia[199];
	RPT_Buffer_hmi.pistone_pistola_1[200] 	:= RPT_Buffer_hmi.pistone_pistola_1[199];
	RPT_Buffer_hmi.pistone_pistola_2[200] 	:= RPT_Buffer_hmi.pistone_pistola_2[199];
	RPT_Buffer_hmi.pistone_soll_su[200] 	:= RPT_Buffer_hmi.pistone_soll_su[199];
	RPT_Buffer_hmi.pistone_soll_giu[200] 	:= RPT_Buffer_hmi.pistone_soll_giu[199];
	RPT_Buffer_hmi.sensore_pistola[200] 	:= RPT_Buffer_hmi.sensore_pistola[199];

END_PROGRAM
```

#### Init.st - Init code
```iecst
PROGRAM _INIT
	(* Insert code here *)

	indice1 := 210;
END_PROGRAM
```

#### Types.typ - Local data types
```iecst
TYPE
	typ_rpt_buffer_hmi : 	STRUCT
		bilancia : ARRAY[1..200]OF REAL := [200(0.0)];
		sensore_pistola : ARRAY[1..200]OF REAL := [200(0.0)];
		pistone_soll_giu : ARRAY[1..200]OF REAL := [200(0.0)];
		pistone_soll_su : ARRAY[1..200]OF REAL := [200(0.0)];
		pistone_pistola_2 : ARRAY[1..200]OF REAL := [200(0.0)];
		pistone_pistola_1 : ARRAY[1..200]OF REAL := [200(0.0)];
		time_stamp : ARRAY[0..249]OF DATE_AND_TIME;
	END_STRUCT;
	typ_rpt_buffer : 	STRUCT
		bilancia : ARRAY[0..249]OF STRING[50] := [250('0')];
		sensore_pistola : ARRAY[0..249]OF USINT := [250(255)];
		pistone_soll_giu : ARRAY[0..249]OF USINT := [250(255)];
		pistone_soll_su : ARRAY[0..249]OF USINT := [250(255)];
		pistone_pistola_2 : ARRAY[0..249]OF USINT := [250(255)];
		pistone_pistola_1 : ARRAY[0..249]OF USINT := [250(255)];
		time_stamp : ARRAY[0..249]OF DATE_AND_TIME;
	END_STRUCT;
END_TYPE
```

#### Variables.var - Local variables
```iecst
VAR
	Test : BOOL := FALSE;
	trend_enable : BOOL := FALSE;
	Bilancia : REAL := 0.0;
	gun_1_b : BOOL := FALSE;
	gun_2_b : BOOL := FALSE;
	i : USINT := 0;
	indice : USINT := 0;
	indice1 : USINT := 0;
	indice2 : USINT := 0;
	k : USINT := 0;
	kk : USINT := 0;
	pistone_pistola_1 : USINT := 0;
	pistone_pistola_2 : USINT := 0;
	pistone_soll_giu : USINT := 0;
	pistone_soll_su : USINT := 0;
	Piston_Up_b : BOOL := FALSE;
	RPT_Buffer : typ_rpt_buffer := (bilancia:=[250('0')],sensore_pistola:=[250(255)],pistone_soll_giu:=[250(255)],pistone_soll_su:=[250(255)],pistone_pistola_2:=[250(255)],pistone_pistola_1:=[250(255)]);
	RPT_Buffer_hmi : typ_rpt_buffer_hmi;
	s01_b : BOOL := FALSE;
	sensore_pistola : USINT := 0;
	Str_Length : INT := 0;
	Str_weight : STRING[80] := '';
	Hmi_trend_03 : HMI_trend;
	Hmi_trend_04 : HMI_trend;
	Hmi_trend_05 : HMI_trend;
	Hmi_trend_06 : HMI_trend;
	Hmi_trend_02 : HMI_trend;
	Hmi_trend_01 : HMI_trend;
	updt_hmi_trend : BOOL := FALSE;
END_VAR
```

#### LocalFunctions.fun
```iecst
{REDUND_ERROR} FUNCTION_BLOCK HMI_trend (*TODO: Add your comment here*) (*$GROUP=User,$CAT=User,$GROUPICON=User.png,$CATICON=User.png*)
	VAR_INPUT
		DataIn : {REDUND_UNREPLICABLE} REAL;
		INOutStatus : {REDUND_UNREPLICABLE} INT;
		INWrite : BOOL;
		INRead : BOOL;
		clear_data : BOOL;
	END_VAR
	VAR_OUTPUT
		DataOut : {REDUND_UNREPLICABLE} REAL;
	END_VAR
	VAR CONSTANT
		BufferMax : INT := 200;
		BufferMin : INT := 1;
	END_VAR
	VAR
		NoOfDataPoints : {REDUND_UNREPLICABLE} INT;
	END_VAR
	VAR_OUTPUT
		Buffer : ARRAY[BufferMin..BufferMax] OF REAL;
	END_VAR
	VAR
		pIn : {REDUND_UNREPLICABLE} INT;
		pOut : {REDUND_UNREPLICABLE} INT;
		p : INT;
	END_VAR
END_FUNCTION_BLOCK
```

#### HMI_rend.st
```iecst
(* TODO: Add your comment here *)
FUNCTION_BLOCK HMI_trend

	IF (pIn = 0) 	THEN pIn	:= BufferMin; END_IF
	IF (pOut = 0) 	THEN pOut	:= BufferMin; END_IF

	// input
	IF (INWrite) THEN
		Buffer[BufferMax] := DataIn; //insert

		IF (Buffer[BufferMax-1] <> -1) THEN
			Buffer[BufferMin] := -1;
			FOR pIn:=BufferMin TO BufferMax-1 DO
				IF (Buffer[pIn] = -1) THEN
					Buffer[pIn] := Buffer[pIn+1];
					Buffer[pIn+1] := -1;
				END_IF
			END_FOR;
		END_IF

		FOR pIn:=BufferMax-1 TO BufferMin BY -1 DO
			IF (Buffer[pIn] = -1) THEN
				Buffer[pIn] := Buffer[pIn+1];
				Buffer[pIn+1] := -1;
			END_IF
		END_FOR;
	END_IF

	// output

	IF (INRead) THEN
		Buffer[BufferMin] := 0;
		FOR pOut:=BufferMin TO BufferMax-1 DO
			IF (Buffer[pOut] = 0) THEN
				Buffer[pOut] := Buffer[pOut+1];
				Buffer[pOut+1] := 0;
			END_IF
		END_FOR;
	END_IF

	DataOut := Buffer[BufferMin]; // out

	IF (clear_data) THEN
		FOR p:=BufferMin TO BufferMax-1 DO
			Buffer[p] := 0;
		END_FOR;
	END_IF

//	//take out data from buffer
//	IF INOutStatus = 2 THEN
//		IF NoOfDataPoints > 0 THEN //there must be data in buffer
//			DataOut := Buffer[pOut];
//			Buffer[pOut] := 0; //set to 0 to show that the value is removed
//			NoOfDataPoints := NoOfDataPoints -1;
//			IF pOut < BufferMax-1 THEN
//				pOut := pOut +1;
//			ELSE
//				pOut := BufferMin;
//			END_IF;
//		END_IF;
//	END_IF;

	//buffer full. last value overwritten, move pIn pointer
//	IF NoOfDataPoints >= BufferMax-1 THEN
////		pIn := pOut;
//		pIn := 6;
//	END_IF;

END_FUNCTION_BLOCK
```

### Program Logical/main/Param_Fix

#### Cyclic.st
```iecst
PROGRAM _CYCLIC
	(* Insert code here *)
	IF Pesi_0.Max_Weight_B < Pesi_0.Min_Weight_B THEN Pesi_0.Max_Weight_B := Pesi_0.Min_Weight_B; END_IF
	IF Pesi_0.Max_Weight_A < Pesi_0.Min_Weight_A THEN Pesi_0.Max_Weight_A := Pesi_0.Min_Weight_A; END_IF
	IF Pesi_0.Min_Weight_B < Pesi_0.Max_Weight_A THEN Pesi_0.Min_Weight_B := Pesi_0.Max_Weight_A; END_IF
END_PROGRAM
```

### Program Logical/main/RPT_CSV (ANSIC)

#### RPT_CSV_Cyclic.c - Cyclic code
```c
/********************************************************************
 * COPYRIGHT --
 ********************************************************************
 * Program: RPT_CSV
 * File: Scrittura_ReportCyclic.c
 * Author: Stefano
 * Created: January 20, 2021
 ********************************************************************
 * CUSTOM CSV REPORT MADE FOR HOUSTON FOAM
 ********************************************************************/

#include <bur/plctypes.h>

#ifdef _DEFAULT_INCLUDES
#include <AsDefault.h>
#endif
#include <asstring.h>
#include <string.h>

#define DENSITA	1
#define MASTER	0

void _CYCLIC RPT_CSV_Cyclic(void)
{
	//data to write
	kgb=0;

	for (kgb = 0; kgb < 30; kgb++)
	{
		rpt_row[kgb]= 1;

	}

	if (!glb_data.Trigger) rpt_write_req = 0;

	if (fucking_debug) step_rpt = step_force;
	switch (step_rpt) /* Stato di idle */
	{
		case WAIT:
		case ERROR:

			if 		(glb_data.Trigger && !rpt_write_req)
			{
				step_rpt = CHECK_FILES_NAME;
				rpt_write_req = 1;				// Resetto la richiesta di scrittura del report
				glb_data.Trigger = 0;			// Machine Cycle done Trigger reset;
			}
			break;;

		case CHECK_FILES_NAME:	// GUARDO SE IL FILE CREATO E' LO STESSO DEL MASTER

			step_rpt = CREATE_FILE_NAME;

			break;;

		case CREATE_FILE_NAME: 	// CREO IL NOME DEI FILE

			memset (&FileCreate_01,          0, sizeof(FileCreate_typ)		);
			memset (&FileWrite_01,           0, sizeof(FileWrite_typ) 		);
			memset (&FileClose_01,           0, sizeof(FileClose_typ) 		);
			memset (&FileCreate_03,          0, sizeof(FileCreate_typ)      );
			memset (&FileOpen_03,            0, sizeof(FileOpen_typ)        );
			memset (&FileWrite_03,           0, sizeof(FileWrite_typ)       );
			memset (&FileClose_03,           0, sizeof(FileClose_typ)		);
			memset (string_rpt,				 '\0', sizeof(string_rpt)		);
			memset (nome_file_doc,			 '\0', sizeof(nome_file_doc)	);
			memset (nome_file_csv,			 '\0', sizeof(nome_file_csv)	);
			memset (support_str,			 '\0', sizeof(support_str)		);
			offset 		= 0;

			/* Trasferisco nella struttura support_str l'orario attuale */
			DT_TO_DTStructure(glb_time, (UDINT)&struct_time);

			/* Genero il nome del file con la data odierna formato YYYY-MM-DD */

			// inserimento anno nel nome del file
			memset (support_str, '\0', sizeof(support_str));
			itoa(struct_time.year, (UDINT)&support_str);
			strcpy(nome_file_doc, support_str);
			strcat(nome_file_doc, "-");

			// inserimento mese nel nome del file
			memset (support_str, '\0', sizeof(support_str));
			itoa(struct_time.month, (UDINT)&support_str);
			if (strlen(support_str) == 1) strcat(nome_file_doc, "0");
			strcat(nome_file_doc, support_str);
			strcat(nome_file_doc, "-");

			// inserimento giorno nel nome del file
			memset (support_str, '\0', sizeof(support_str));
			itoa(struct_time.day, (UDINT)&support_str);
			if (strlen(support_str) == 1) strcat(nome_file_doc, "0");
			strcat(nome_file_doc, support_str);
			strcat(nome_file_doc, "-");

//			// inserimento nome ricetta nel nome del file
//			memset (support_str, '\0', sizeof(support_str));
//			strcat(support_str, glb_ultima_ricetta);
//			if (strlen(support_str) == 1) strcat(nome_file_doc, "0");
//			strcat(nome_file_doc, support_str);

			strcpy(nome_file_csv, nome_file_doc);
			strcat(nome_file_csv, ".csv");				// creo il file YYYY-MM-DD.csv

			step_rpt = CREATE_CSV_FILE;

			break;;

		case CREATE_CSV_FILE: // CREO IL FILE .CSV

			FileCreate_03.enable  = 1;
			FileCreate_03.pDevice = (UDINT) "DATA";
			FileCreate_03.pFile   = (UDINT) &nome_file_csv;

			FileCreate(&FileCreate_03);

			if (FileCreate_03.status == 0)
			{
				offset 					= 0;
				step_rpt   					= OPEN_CSV_FILE;
				FileCreate_03.enable 	= 0;
				RowCounterFile			= 0;
			}
			else if (FileCreate_03.status == 20705) /* file già esistente */
			{
				step_rpt 					= OPEN_CSV_FILE;
				FileCreate_03.status 	= 0;
				FileCreate_03.enable 	= 0;
			}

			break;;

		case OPEN_CSV_FILE: // APRO IL FILE CSV

			FileOpen_03.enable    = 1;
			FileOpen_03.pDevice   = (UDINT) "DATA";
			FileOpen_03.pFile     = (UDINT) &nome_file_csv;
			FileOpen_03.mode      = FILE_RW;

			FileOpen(&FileOpen_03);

			if (FileOpen_03.status == 0)
			{
				step_rpt = CREATE_HEADER_CSV_FILE;

				memset (string_rpt, '\0', sizeof(string_rpt));
				memset (support_str,   '\0', sizeof(support_str)  );

				FileOpen_03.status 	= 0;
				ident_csv			= FileOpen_03.ident;
				FileOpen_03.enable 	= 0;
			}
			else if (FileOpen_03.status != 65535)
			{
				step_rpt	 			= ERROR;
				numero_errore   	= FileIoGetSysError();
				FileOpen_03.enable = 0;
			}

			break;;

		// Chiamato dal master
		case CREATE_HEADER_CSV_FILE:

			// Il file è vuoto
			if (FileOpen_03.filelen < 101) //lunghezza della intestazione
			{
				// HEADER CDV FILE -------------------------------------------------------------------
				// Salvo l'intestazione di 120 caratteri

				//	sep=;
				//	Report
				//	Dati misurazione particolari
				//	Mould Code = jhgfdsasdfghj;
				//
				//	Timestamp;Recipe Name;QRCode;Dato 1;Dato 2;Dato 3;Dato 4;Dato 5;Dato 6;Dato 7;Dato 8;Code;Material type;Material Color;Mould Code;Density;Volume;Peso;Temperature;Peso inserto;\n
				//  Timestamp;Recipe Name;QRCode;Dato 1;Dato 2;Dato 3;Dato 4;Dato 5;Dato 6;Dato 7;Dato 8;Code;Material type;Material Color;Mould Code;Density;Volume;Peso;Temperature;Peso inserto;\n
				//  012345678901234567890123456789012345678901234567890123456789012345678901234567890123456789012345678901234567890123456789
				//	0_________1_________2_________3_________4_________5_________6_________7_________8_________9_________10________11________

				strcpy(string_rpt, "sep=;\nReport\nDati misurazione particolari\n\n");
				strcat(string_rpt, "\n");
//				strcat(string_rpt, "Timestamp;Recipe Name;QRCode;Dato 1;Dato 2;Dato 3;Dato 4;Dato 5;Dato 6;Dato 7;Dato 8;Code;Material type;Material Color;Mould Code;Density;Volume;Peso;Temperature;Peso inserto;");
				strcat(string_rpt, "Timestamp;Recipe Name;QRCode;");

				strcat(string_rpt, "\n");
				// END HEADER ------------------------------------------------------------------------

				// TIMESTAMP
				memset (support_str, '\0', sizeof(support_str));
				ascDT(glb_data.time_stamp[xxx],(UDINT)&support_str,sizeof(support_str));
				if (strlen(support_str) == 1) strcat(string_rpt, "0");
				strcat(string_rpt, support_str);
				strcat(string_rpt, ";");

				// BILANCIA
				memset (support_str, '\0', sizeof(support_str));
				strcat(string_rpt, glb_data.bilancia[xxx]);
				strcat(string_rpt, ";");

				// SENSORE PISTOLA
				memset (support_str, '\0', sizeof(support_str));
				itoa(glb_data.sensore_pistola[xxx], (UDINT)&support_str);
				strcat(string_rpt, support_str);
				strcat(string_rpt, ";");

				// PISTONE SOLLEVAMENTO SU 1
				memset (support_str, '\0', sizeof(support_str));
				itoa(glb_data.pistone_soll_su[xxx], (UDINT)&support_str);
				strcat(string_rpt, support_str);
				strcat(string_rpt, ";");

				// PISTONE SOLLEVAMENTO GIU 1
				memset (support_str, '\0', sizeof(support_str));
				itoa(glb_data.pistone_soll_giu[xxx], (UDINT)&support_str);
				strcat(string_rpt, support_str);
				strcat(string_rpt, ";");

				// PISTOLA 1
				memset (support_str, '\0', sizeof(support_str));
				itoa(glb_data.pistone_pistola_1[xxx], (UDINT)&support_str);
				strcat(string_rpt, support_str);
				strcat(string_rpt, ";");

				// PISTOLA 1
				memset (support_str, '\0', sizeof(support_str));
				itoa(glb_data.pistone_pistola_1[xxx], (UDINT)&support_str);
				strcat(string_rpt, support_str);
				strcat(string_rpt, ";");

				// PISTOLA 2
				memset (support_str, '\0', sizeof(support_str));
				itoa(glb_data.pistone_pistola_2[xxx], (UDINT)&support_str);
				strcat(string_rpt, support_str);
				strcat(string_rpt, ";");

				strcat(string_rpt, "\n");

				filelen = 0;
				str_lenght = strlen(string_rpt); /* restituisce la lunghezza della stringa senza terminatore nullo */

				/* Preparo la struttura per la funzione di scrittura */
				FileWrite_03.enable   = 1;
				FileWrite_03.ident    = ident_csv;
				FileWrite_03.offset   = filelen;
				FileWrite_03.pSrc     = (UDINT) &string_rpt[0];
				//FileWrite_03.len      =	sizeof(USINT) * 240;
				FileWrite_03.len      =	str_lenght;
				offset                = sizeof(USINT) * 240;

				RowCounterFile		  = 2; //2 ROWS * 110 BYTES

				step_rpt = WRITE_CSV_FILE;
			}
			else if (FileOpen_03.filelen > 120) // Il file è già stato scritto
			{

				// TIMESTAMP
				memset (support_str, '\0', sizeof(support_str));
				ascDT(glb_data.time_stamp[xxx],(UDINT)&support_str,sizeof(support_str));
				if (strlen(support_str) == 1) strcat(string_rpt, "0");
				strcat(string_rpt, support_str);
				strcat(string_rpt, ";");

				// BILANCIA
				memset (support_str, '\0', sizeof(support_str));
				strcat(string_rpt, glb_data.bilancia[xxx]);
				strcat(string_rpt, ";");

				// SENSORE PISTOLA
				memset (support_str, '\0', sizeof(support_str));
				itoa(glb_data.sensore_pistola[xxx], (UDINT)&support_str);
				strcat(string_rpt, support_str);
				strcat(string_rpt, ";");

				// PISTONE SOLLEVAMENTO SU 1
				memset (support_str, '\0', sizeof(support_str));
				itoa(glb_data.pistone_soll_su[xxx], (UDINT)&support_str);
				strcat(string_rpt, support_str);
				strcat(string_rpt, ";");

				// PISTONE SOLLEVAMENTO GIU 1
				memset (support_str, '\0', sizeof(support_str));
				itoa(glb_data.pistone_soll_giu[xxx], (UDINT)&support_str);
				strcat(string_rpt, support_str);
				strcat(string_rpt, ";");

				// PISTOLA 1
				memset (support_str, '\0', sizeof(support_str));
				itoa(glb_data.pistone_pistola_1[xxx], (UDINT)&support_str);
				strcat(string_rpt, support_str);
				strcat(string_rpt, ";");

				// PISTOLA 1
				memset (support_str, '\0', sizeof(support_str));
				itoa(glb_data.pistone_pistola_1[xxx], (UDINT)&support_str);
				strcat(string_rpt, support_str);
				strcat(string_rpt, ";");

				// PISTOLA 2
				memset (support_str, '\0', sizeof(support_str));
				itoa(glb_data.pistone_pistola_2[xxx], (UDINT)&support_str);
				strcat(string_rpt, support_str);
				strcat(string_rpt, ";");

				strcat(string_rpt, "\n");

				RowCounterFile++;
				filelen = RowCounterFile * 120;
				filelen = FileOpen_03.filelen;

				str_lenght = strlen(string_rpt); /* restituisce la lunghezza della stringa senza terminatore nullo */

				/* Preparo la struttura per la funzione di scrittura */
				FileWrite_03.enable   = 1;
				FileWrite_03.ident    = ident_csv;
				FileWrite_03.offset   = filelen;
				FileWrite_03.pSrc     = (UDINT) &string_rpt[0];
				//FileWrite_03.len      =	sizeof(USINT) * 120;
				FileWrite_03.len      =	str_lenght;
				offset               += sizeof(USINT) * 120;

				step_rpt = WRITE_CSV_FILE;
			}
			else  // Chiamato dal controllo densità con numero di ciclo a 0
			{
				step_rpt = CLOSE_CSV_FILE;
			}

			break;

		case WRITE_CSV_FILE:

			FileWrite(&FileWrite_03);

			if (FileWrite_03.status == 0)
			{
				//glb_comandi.cmd_scrivi_report 	= 0;					// Resetto la richiesta di scrittura del report
				//rpt_write_req				 	= 0;
				glb_data.Report_recorded 		= 1;
				step_rpt 						  	= CLOSE_CSV_FILE;
				FileWrite_03.enable 		  	= 0;
			}
			else if (FileWrite_03.status != 65535)
			{
				step_rpt	 			= CLOSE_CSV_FILE;
				numero_errore   	= FileIoGetSysError();
				FileWrite_03.enable = 0;
			}

			break;;

		case CLOSE_CSV_FILE:

			FileClose_03.enable = 1;
			FileClose_03.ident  = ident_csv;
			//rpt_write_req				 	= 0;

			FileClose(&FileClose_03);

			if (FileClose_03.status == 0)
			{
				step_rpt 				= WAIT;
				FileClose_03.enable = 0;
			}
			else if (FileClose_03.status != 65535)
			{
				step_rpt	 			= WAIT;
				numero_errore   	= FileIoGetSysError();
				FileClose_03.enable = 0;
			}

			break;;
	}

	/*********************************************** CREATE DIR WHERE SAVE THE CAVITIES INFO LINKE TO THE RECIPES **************************************************/

	if ((DirCreate_05.status == 0) ||  (DirCreate_05.status == 20725))	    /* if status ok (0) or dir already exists (20725)		 	*/
	{
		DirCreate_05.enable 	= 0;
	}

}
```

#### RPT_CSV_Init.c - Initialization code
```c
#include <bur/plctypes.h>
#include <string.h>

#ifdef _DEFAULT_INCLUDES
#include <AsDefault.h>
#endif

void _INIT RPT_CSV_Init(void)
{
	/* Pulisco la memoria */
	memset (&DirCreate_03,			 0, sizeof(DirCreate_typ)   );
	memset (&DirCreate_05,			 0, sizeof(DirCreate_typ)   );
	memset (&FileCreate_01,          0, sizeof(FileCreate_typ)  );
	memset (&FileCreate_03,          0, sizeof(FileCreate_typ)  );
	memset (&FileOpen_03,            0, sizeof(FileOpen_typ)    );
	memset (&FileWrite_01,           0, sizeof(FileWrite_typ)   );
	memset (&FileWrite_03,           0, sizeof(FileWrite_typ)   );
	memset (&FileClose_01,           0, sizeof(FileClose_typ)	);
	memset (&FileClose_03,           0, sizeof(FileClose_typ)	);
	memset (string_rpt,				'\0', 	sizeof(string_rpt)  	);
	memset (support_str,			'\0', 	sizeof(support_str)    );
	step_rpt = WAIT;
	RowCounterFile				= 0;

	DirCreate_03.enable  = 1;
	DirCreate_03.pDevice = (UDINT) "CF";
	DirCreate_03.pName   = (UDINT) "DATA";

	DirCreate(&DirCreate_03);

	if ((DirCreate_03.status == 0) ||  (DirCreate_03.status == 20725))	    /* if status ok (0) or dir already exists (20725)		 		*/
	{
		DirCreate_03.status = 0;															/* set status ok											*/
	}

	DirCreate_05.enable  = 1;
	DirCreate_05.pDevice = (UDINT) "CF";
	DirCreate_05.pName   = (UDINT) "CFG";

	DirCreate(&DirCreate_05);

	if ((DirCreate_05.status == 0) ||  (DirCreate_05.status == 20725))	    /* if status ok (0) or dir already exists (20725)		 		*/
	{
		DirCreate_05.status = 0;															/* set status ok											*/
	}
//	rt_info.enable = 1;     /* enables the function */
//	RTInfo(&rt_info);       /* gets information from the software object */
//	sys_info.enable = 1;    /* enables the function */
//	SysInfo(&sys_info);     /* gets information from the system */
}
```

#### Types.typ - Local data types
```iecst
TYPE
	Enum_Step :
		(
		WAIT := 0, (*ATTESA*)
		CHECK_FILES_NAME := 1, (*CONTROLLO_NOMI_FILES*)
		CREATE_FILE_NAME := 2, (*CREO_NOMI_FILE*)
		DELETE_DOC_FILE := 3, (*ELIMINO_FILE_DOC*)
		CREATE_DOC_FILE := 4, (*CREO_FILE_DOC*)
		PREPARE_DOC_FILE := 5, (*PREPARO_FILE_DOC*)
		WRITE_DOC_FILE := 6, (*SCRIVO_FILE_DOC*)
		CLOSE_DOC_FILE := 7, (*CHIUDO_FILE_DOC*)
		CREATE_CSV_FILE := 8, (*CREO_FILE_CSV*)
		OPEN_CSV_FILE := 9, (*APRO_FILE_CSV*)
		CREATE_HEADER_CSV_FILE := 10, (*PREPARO_FILE_CSV*)
		WRITE_CSV_FILE := 11, (*SCRIVO_FILE_CSV*)
		CLOSE_CSV_FILE := 12, (*CHIUDO_FILE_CSV*)
		ERROR := 13 (*ERRORE*)
		);
	typAlarmHistory : 	STRUCT
		id : UDINT;
		description : STRING[80];
	END_STRUCT;
END_TYPE
```

#### Variables.var - Local variables
```iecst
VAR
	xxx : USINT := 0;
	glb_MacCycleDoneTrigg : BOOL;
	CmdAckError_0 : BOOL;
	DirCreate_03 : DirCreate;
	DirCreate_05 : DirCreate;
	DTGetTime_1 : DTGetTime;
	FDelete : FileDelete;
	FileClose_01 : FileClose;
	FileClose_03 : FileClose;
	FileCreate_01 : FileCreate;
	FileCreate_03 : FileCreate;
	filelen : UDINT; (*Dove inserire la riga da scrivere sul file csv*)
	FileOpen_03 : FileOpen;
	FileWrite_01 : FileWrite;
	FileWrite_03 : FileWrite;
	fucking_debug : BOOL;
	ident_csv : UDINT; (*fucking identification file (the famous HANDLE)*)
	ident_doc : UDINT;
	kgb : UINT;
	nome_file_csv : STRING[32];
	nome_file_doc : STRING[32];
	note : STRING[61]; (*Eventuali note da allegare*)
	numero_errore : UINT; (*Numero dell'errore delle funzioni di I/O*)
	offset : UDINT; (*Numero di byte scritti su CSV*)
	RowCounterFile : UDINT;
	rpt_row : ARRAY[0..29] OF USINT;
	rpt_write_req : BOOL;
	step_rpt : USINT;
	step_force : USINT;
	step_recipe : USINT; (*was step (Recipes)*)
	rpt_name : STRING[30];
	string_rpt2 : STRING[500];
	string_rpt : STRING[1500];
	rptMpRecipeInfo : STRING[200];
	struct_time : DTStructure; (*Struttura dove converto la data della commessa*)
	str_lenght : UDINT;
	supp : REAL;
	support_str1 : STRING[40];
	support_str : STRING[40];
	j : USINT; (*counter*)
END_VAR
```

### Program Logical/main/RPT_CSV_ST

#### Variables.var
```iecst
VAR
	New_CSV_cmd : BOOL := FALSE;
	Counter_Reset : BOOL := FALSE;
	Day_test : USINT := 0;
END_VAR
VAR RETAIN
	Saved_day : USINT := 0;
END_VAR
VAR
	New_CSV : BOOL := FALSE;
END_VAR
VAR RETAIN
	Counter : USINT := 0;
END_VAR
VAR
	TP_01 : TP := (0);
	estensione : STRING[80] := '.csv';
	space : STRING[80] := '-';
	CFG : STRING[80] := 'CFG';
	DATA : STRING[80] := 'DATA';
	CF : STRING[80] := 'CF';
	xxx : USINT := 0;
	glb_MacCycleDoneTrigg : BOOL;
	CmdAckError_0 : BOOL;
	DirCreate_03 : DirCreate;
	DirCreate_05 : DirCreate;
	DTGetTime_1 : DTGetTime;
	FDelete : FileDelete;
	FileClose_01 : FileClose;
	FileClose_03 : FileClose;
	FileCreate_01 : FileCreate;
	FileCreate_03 : FileCreate;
	filelen : UDINT; (*Dove inserire la riga da scrivere sul file csv*)
	FileOpen_03 : FileOpen;
	FileWrite_01 : FileWrite;
	FileWrite_03 : FileWrite;
	fucking_debug : BOOL;
	ident_csv : UDINT; (*fucking identification file (the famous HANDLE)*)
	ident_doc : UDINT;
	kgb : UINT;
	nome_file_csv : STRING[32];
	nome_file_doc : STRING[32];
	note : STRING[61]; (*Eventuali note da allegare*)
	numero_errore : UINT; (*Numero dell'errore delle funzioni di I/O*)
	offset : UDINT; (*Numero di byte scritti su CSV*)
	RowCounterFile : UDINT;
	rpt_row : ARRAY[0..29] OF USINT;
	rpt_write_req : BOOL;
	step_rpt : Enum_Step;
	step_force : USINT;
	step_recipe : USINT; (*was step (Recipes)*)
	rpt_name : STRING[30];
	string_rpt2 : STRING[500];
	string_rpt : STRING[1500];
	rptMpRecipeInfo : STRING[200];
	struct_time : DTStructure; (*Struttura dove converto la data della commessa*)
	str_lenght : UDINT;
	supp : REAL;
	support_str1 : STRING[40];
	support_str : STRING[40];
	j : USINT; (*counter*)
END_VAR
```
